LIN {X 0,Y 516.961,Z 452.089,A -85,B 0,C 180,E1 -4941.399,E2 -4941.399} C_VEL
LIN {X 0,Y 517.016,Z 452.086,A -85,B 0,C 180,E1 -4943.757,E2 -4943.757} C_VEL
LIN {X 0,Y 517.09,Z 452.073,A -85,B 0,C 180,E1 -4947.663,E2 -4947.663} C_VEL
LIN {X 0,Y 517.099,Z 452.072,A -85,B 0,C 180,E1 -4950.779,E2 -4950.779} C_VEL
LIN {X 0,Y 517.016,Z 452.086,A -85,B 0,C 180,E1 -4953.117,E2 -4953.117} C_VEL
LIN {X 0,Y 516.993,Z 452.088,A -85,B 0,C 180,E1 -4956.243,E2 -4956.243} C_VEL
LIN {X 0,Y 516.975,Z 452.088,A -85,B 0,C 180,E1 -4958.6,E2 -4958.6} C_VEL
LIN {X 0,Y 516.958,Z 452.09,A -85,B 0,C 180,E1 -4961.807,E2 -4961.807} C_VEL
LIN {X 0,Y 516.951,Z 452.092,A -85,B 0,C 180,E1 -4965.146,E2 -4965.146} C_VEL
LIN {X 0,Y 516.93,Z 452.096,A -85,B 0,C 180,E1 -4968.222,E2 -4968.222} C_VEL
LIN {X 0,Y 516.917,Z 452.093,A -85,B 0,C 180,E1 -4970.701,E2 -4970.701} C_VEL
LIN {X 0,Y 516.909,Z 452.096,A -85,B 0,C 180,E1 -4974.072,E2 -4974.072} C_VEL
LIN {X 0,Y 516.927,Z 452.095,A -85,B 0,C 180,E1 -4976.658,E2 -4976.658} C_VEL
LIN {X 0,Y 516.916,Z 452.1,A -85,B 0,C 180,E1 -4979.523,E2 -4979.523} C_VEL
LIN {X 0,Y 516.9,Z 452.1,A -85,B 0,C 180,E1 -4982.543,E2 -4982.543} C_VEL
LIN {X 0,Y 516.883,Z 452.099,A -85,B 0,C 180,E1 -4985.331,E2 -4985.331} C_VEL
LIN {X 0,Y 516.884,Z 452.099,A -85,B 0,C 180,E1 -4987.943,E2 -4987.943} C_VEL
LIN {X 0,Y 516.886,Z 452.1,A -85,B 0,C 180,E1 -4990.741,E2 -4990.741} C_VEL
LIN {X 0,Y 516.887,Z 452.097,A -85,B 0,C 180,E1 -4992.831,E2 -4992.831} C_VEL
LIN {X 0,Y 516.926,Z 452.097,A -85,B 0,C 180,E1 -4995.01,E2 -4995.01} C_VEL
LIN {X 0,Y 516.919,Z 452.096,A -85,B 0,C 180,E1 -4998.398,E2 -4998.398} C_VEL
LIN {X 0,Y 516.883,Z 452.103,A -85,B 0,C 180,E1 -5001.284,E2 -5001.284} C_VEL
LIN {X 0,Y 516.892,Z 452.102,A -85,B 0,C 180,E1 -5004.221,E2 -5004.221} C_VEL
LIN {X 0,Y 516.899,Z 452.097,A -85,B 0,C 180,E1 -5007.053,E2 -5007.053} C_VEL
LIN {X 0,Y 516.895,Z 452.098,A -85,B 0,C 180,E1 -5009.796,E2 -5009.796} C_VEL
LIN {X 0,Y 516.931,Z 452.095,A -85,B 0,C 180,E1 -5012.467,E2 -5012.467} C_VEL
LIN {X 0,Y 516.911,Z 452.097,A -85,B 0,C 180,E1 -5015.072,E2 -5015.072} C_VEL
LIN {X 0,Y 516.888,Z 452.101,A -85,B 0,C 180,E1 -5018.462,E2 -5018.462} C_VEL
LIN {X 0,Y 516.904,Z 452.096,A -85,B 0,C 180,E1 -5020.955,E2 -5020.955} C_VEL
LIN {X 0,Y 516.916,Z 452.097,A -85,B 0,C 180,E1 -5023.41,E2 -5023.41} C_VEL
LIN {X 0,Y 516.898,Z 452.099,A -85,B 0,C 180,E1 -5025.833,E2 -5025.833} C_VEL
LIN {X 0,Y 516.967,Z 452.088,A -85,B 0,C 180,E1 -5028.233,E2 -5028.233} C_VEL
LIN {X 0,Y 516.971,Z 452.089,A -85,B 0,C 180,E1 -5031.399,E2 -5031.399} C_VEL
LIN {X 0,Y 517.012,Z 452.086,A -85,B 0,C 180,E1 -5033.757,E2 -5033.757} C_VEL
LIN {X 0,Y 517.084,Z 452.075,A -85,B 0,C 180,E1 -5037.663,E2 -5037.663} C_VEL
LIN {X 0,Y 517.095,Z 452.073,A -85,B 0,C 180,E1 -5040.779,E2 -5040.779} C_VEL
LIN {X 0,Y 517.014,Z 452.084,A -85,B 0,C 180,E1 -5043.117,E2 -5043.117} C_VEL
LIN {X 0,Y 517.011,Z 452.086,A -85,B 0,C 180,E1 -5046.243,E2 -5046.243} C_VEL
LIN {X 0,Y 516.952,Z 452.093,A -85,B 0,C 180,E1 -5049.389,E2 -5049.389} C_VEL
LIN {X 0,Y 516.953,Z 452.09,A -85,B 0,C 180,E1 -5051.807,E2 -5051.807} C_VEL
LIN {X 0,Y 516.946,Z 452.091,A -85,B 0,C 180,E1 -5055.146,E2 -5055.146} C_VEL
LIN {X 0,Y 516.926,Z 452.093,A -85,B 0,C 180,E1 -5058.222,E2 -5058.222} C_VEL
LIN {X 0,Y 516.914,Z 452.099,A -85,B 0,C 180,E1 -5060.701,E2 -5060.701} C_VEL
LIN {X 0,Y 516.912,Z 452.095,A -85,B 0,C 180,E1 -5064.072,E2 -5064.072} C_VEL
LIN {X 0,Y 516.927,Z 452.096,A -85,B 0,C 180,E1 -5066.658,E2 -5066.658} C_VEL
LIN {X 0,Y 516.912,Z 452.097,A -85,B 0,C 180,E1 -5069.524,E2 -5069.524} C_VEL
LIN {X 0,Y 516.896,Z 452.097,A -85,B 0,C 180,E1 -5072.543,E2 -5072.543} C_VEL
LIN {X 0,Y 516.882,Z 452.099,A -85,B 0,C 180,E1 -5075.332,E2 -5075.332} C_VEL
LIN {X 0,Y 516.881,Z 452.1,A -85,B 0,C 180,E1 -5077.943,E2 -5077.943} C_VEL
LIN {X 0,Y 516.886,Z 452.102,A -85,B 0,C 180,E1 -5080.742,E2 -5080.742} C_VEL
LIN {X 0,Y 516.906,Z 452.097,A -85,B 0,C 180,E1 -5082.829,E2 -5082.829} C_VEL
LIN {X 0,Y 516.882,Z 452.102,A -85,B 0,C 180,E1 -5086.107,E2 -5086.107} C_VEL
LIN {X 0,Y 516.916,Z 452.1,A -85,B 0,C 180,E1 -5088.399,E2 -5088.399} C_VEL
LIN {X 0,Y 516.905,Z 452.247,A -85,B 0,C 180,E1 -5091.286,E2 -5091.286} C_VEL
LIN {X 0,Y 518.028,Z 458.682,A -85,B 0,C 180,E1 -5093.832,E2 -5093.832} C_VEL
LIN {X 0,Y 518.109,Z 462.545,A -85,B 0,C 180,E1 -5095.27,E2 -5095.27} C_VEL
LIN {X 0,Y 517.824,Z 470.311,A -85,B 0,C 180,E1 -5098.041,E2 -5098.041} C_VEL
LIN {X 0,Y 517.528,Z 478.131,A -85,B 0,C 180,E1 -5100.733,E2 -5100.733} C_VEL
LIN {X 0,Y 517.309,Z 486.015,A -85,B 0,C 180,E1 -5103.364,E2 -5103.364} C_VEL
LIN {X 0,Y 517.111,Z 493.954,A -85,B 0,C 180,E1 -5105.938,E2 -5105.938} C_VEL
LIN {X 0,Y 516.893,Z 503.251,A -85,B 0,C 180,E1 -5108.881,E2 -5108.881} C_VEL
LIN {X 0,Y 516.737,Z 512.695,A -85,B 0,C 180,E1 -5111.771,E2 -5111.771} C_VEL
LIN {X 0,Y 516.643,Z 522.297,A -85,B 0,C 180,E1 -5114.658,E2 -5114.658} C_VEL
LIN {X 0,Y 516.586,Z 527.093,A -85,B 0,C 180,E1 -5116.101,E2 -5116.101} C_VEL
LIN {X 0,Y 518.446,Z 540.212,A -85,B 0,C 180,E1 -5116.452,E2 -5116.452} C_VEL
LIN {X 0,Y 518.207,Z 553.337,A -85,B 0,C 180,E1 -5116.92,E2 -5116.92} C_VEL
LIN {X 0,Y 517.922,Z 565.66,A -85,B 0,C 180,E1 -5117.527,E2 -5117.527} C_VEL
LIN {X 0,Y 517.632,Z 577.009,A -85,B 0,C 180,E1 -5118.249,E2 -5118.249} C_VEL
LIN {X 0,Y 517.298,Z 588.004,A -85,B 0,C 180,E1 -5119.135,E2 -5119.135} C_VEL
LIN {X 0,Y 517.017,Z 596.964,A -85,B 0,C 180,E1 -5120.02,E2 -5120.02} C_VEL
LIN {X 0,Y 516.772,Z 606.702,A -85,B 0,C 180,E1 -5121.199,E2 -5121.199} C_VEL
LIN {X 0,Y 516.562,Z 614.456,A -85,B 0,C 180,E1 -5122.377,E2 -5122.377} C_VEL
LIN {X 0,Y 516.426,Z 621.601,A -85,B 0,C 180,E1 -5123.75,E2 -5123.75} C_VEL
LIN {X 0,Y 516.314,Z 626.35,A -85,B 0,C 180,E1 -5124.924,E2 -5124.924} C_VEL
LIN {X 0,Y 516.354,Z 629.957,A -85,B 0,C 180,E1 -5126.098,E2 -5126.098} C_VEL
LIN {X 0,Y 516.282,Z 631.807,A -85,B 0,C 180,E1 -5126.879,E2 -5126.879} C_VEL
LIN {X 0,Y 516.26,Z 633.192,A -85,B 0,C 180,E1 -5127.66,E2 -5127.66} C_VEL
LIN {X 0,Y 516.16,Z 634.785,A -85,B 0,C 180,E1 -5129.22,E2 -5129.22} C_VEL
LIN {X 0,Y 516.154,Z 635,A -85,B 0,C 180,E1 -5130,E2 -5130} C_VEL
LIN {X 0,Y 516.192,Z 634.183,A -85,B 0,C 180,E1 -5131.561,E2 -5131.561} C_VEL
LIN {X 0,Y 516.26,Z 633.195,A -85,B 0,C 180,E1 -5132.341,E2 -5132.341} C_VEL
LIN {X 0,Y 516.282,Z 631.81,A -85,B 0,C 180,E1 -5133.122,E2 -5133.122} C_VEL
LIN {X 0,Y 516.344,Z 628.89,A -85,B 0,C 180,E1 -5134.293,E2 -5134.293} C_VEL
LIN {X 0,Y 516.405,Z 624.912,A -85,B 0,C 180,E1 -5135.467,E2 -5135.467} C_VEL
LIN {X 0,Y 516.479,Z 618.961,A -85,B 0,C 180,E1 -5136.798,E2 -5136.798} C_VEL
LIN {X 0,Y 516.641,Z 612.011,A -85,B 0,C 180,E1 -5138.015,E2 -5138.015} C_VEL
LIN {X 0,Y 516.844,Z 603.643,A -85,B 0,C 180,E1 -5139.194,E2 -5139.194} C_VEL
LIN {X 0,Y 517.058,Z 595.052,A -85,B 0,C 180,E1 -5140.178,E2 -5140.178} C_VEL
LIN {X 0,Y 517.417,Z 584.448,A -85,B 0,C 180,E1 -5141.161,E2 -5141.161} C_VEL
LIN {X 0,Y 517.697,Z 572.571,A -85,B 0,C 180,E1 -5142.043,E2 -5142.043} C_VEL
LIN {X 0,Y 518.031,Z 560.478,A -85,B 0,C 180,E1 -5142.736,E2 -5142.736} C_VEL
LIN {X 0,Y 518.274,Z 547.989,A -85,B 0,C 180,E1 -5143.278,E2 -5143.278} C_VEL
LIN {X 0,Y 518.222,Z 537.911,A -85,B 0,C 180,E1 -5143.604,E2 -5143.604} C_VEL
LIN {X 0,Y 516.569,Z 526.747,A -85,B 0,C 180,E1 -5143.899,E2 -5143.899} C_VEL
LIN {X 0,Y 516.624,Z 517.508,A -85,B 0,C 180,E1 -5146.6,E2 -5146.6} C_VEL
LIN {X 0,Y 516.753,Z 507.736,A -85,B 0,C 180,E1 -5149.464,E2 -5149.464} C_VEL
LIN {X 0,Y 516.902,Z 498.047,A -85,B 0,C 180,E1 -5152.398,E2 -5152.398} C_VEL
LIN {X 0,Y 517.068,Z 488.591,A -85,B 0,C 180,E1 -5155.35,E2 -5155.35} C_VEL
LIN {X 0,Y 517.247,Z 480.584,A -85,B 0,C 180,E1 -5157.972,E2 -5157.972} C_VEL
LIN {X 0,Y 517.581,Z 471.425,A -85,B 0,C 180,E1 -5161.191,E2 -5161.191} C_VEL
LIN {X 0,Y 517.951,Z 463.912,A -85,B 0,C 180,E1 -5164.137,E2 -5164.137} C_VEL
LIN {X 0,Y 518.131,Z 460.415,A -85,B 0,C 180,E1 -5165.68,E2 -5165.68} C_VEL
LIN {X 0,Y 517.729,Z 456.632,A -85,B 0,C 180,E1 -5167.652,E2 -5167.652} C_VEL
LIN {X 0,Y 517.139,Z 453.466,A -85,B 0,C 180,E1 -5169.698,E2 -5169.698} C_VEL
LIN {X 0,Y 516.906,Z 452.169,A -85,B 0,C 180,E1 -5170.74,E2 -5170.74} C_VEL
LIN {X 0,Y 516.886,Z 452.103,A -85,B 0,C 180,E1 -5173.903,E2 -5173.903} C_VEL
LIN {X 0,Y 516.886,Z 452.103,A -85,B 0,C 180,E1 -5176.107,E2 -5176.107} C_VEL
LIN {X 0,Y 516.921,Z 452.099,A -85,B 0,C 180,E1 -5178.398,E2 -5178.398} C_VEL
LIN {X 0,Y 516.886,Z 452.103,A -85,B 0,C 180,E1 -5181.284,E2 -5181.284} C_VEL
LIN {X 0,Y 516.85,Z 452.296,A -85,B 0,C 180,E1 -5184.218,E2 -5184.218} C_VEL
LIN {X 0,Y 516.898,Z 453.753,A -85,B 0,C 180,E1 -5186.12,E2 -5186.12} C_VEL
LIN {X 0,Y 516.776,Z 456.139,A -85,B 0,C 180,E1 -5188.958,E2 -5188.958} C_VEL
LIN {X 0,Y 516.644,Z 458.463,A -85,B 0,C 180,E1 -5191.568,E2 -5191.568} C_VEL
LIN {X 0,Y 516.58,Z 460.901,A -85,B 0,C 180,E1 -5194.192,E2 -5194.192} C_VEL
LIN {X 0,Y 516.473,Z 463.37,A -85,B 0,C 180,E1 -5196.758,E2 -5196.758} C_VEL
LIN {X 0,Y 516.437,Z 466.473,A -85,B 0,C 180,E1 -5199.884,E2 -5199.884} C_VEL
LIN {X 0,Y 516.371,Z 469.198,A -85,B 0,C 180,E1 -5202.577,E2 -5202.577} C_VEL
LIN {X 0,Y 516.369,Z 471.797,A -85,B 0,C 180,E1 -5205.093,E2 -5205.093} C_VEL
LIN {X 0,Y 516.313,Z 473.008,A -85,B 0,C 180,E1 -5206.219,E2 -5206.219} C_VEL
LIN {X 0,Y 518.436,Z 484.731,A -85,B 0,C 180,E1 -5206.601,E2 -5206.601} C_VEL
LIN {X 0,Y 518.175,Z 497.984,A -85,B 0,C 180,E1 -5207.118,E2 -5207.118} C_VEL
LIN {X 0,Y 517.895,Z 510.399,A -85,B 0,C 180,E1 -5207.785,E2 -5207.785} C_VEL
LIN {X 0,Y 517.609,Z 521.398,A -85,B 0,C 180,E1 -5208.546,E2 -5208.546} C_VEL
LIN {X 0,Y 517.289,Z 531.681,A -85,B 0,C 180,E1 -5209.431,E2 -5209.431} C_VEL
LIN {X 0,Y 517.006,Z 540.914,A -85,B 0,C 180,E1 -5210.414,E2 -5210.414} C_VEL
LIN {X 0,Y 516.778,Z 549.836,A -85,B 0,C 180,E1 -5211.594,E2 -5211.594} C_VEL
LIN {X 0,Y 516.576,Z 557.015,A -85,B 0,C 180,E1 -5212.771,E2 -5212.771} C_VEL
LIN {X 0,Y 516.474,Z 561.855,A -85,B 0,C 180,E1 -5213.75,E2 -5213.75} C_VEL
LIN {X 0,Y 516.314,Z 566.555,A -85,B 0,C 180,E1 -5214.924,E2 -5214.924} C_VEL
LIN {X 0,Y 516.373,Z 570.142,A -85,B 0,C 180,E1 -5216.098,E2 -5216.098} C_VEL
LIN {X 0,Y 516.283,Z 572.001,A -85,B 0,C 180,E1 -5216.879,E2 -5216.879} C_VEL
LIN {X 0,Y 516.261,Z 573.402,A -85,B 0,C 180,E1 -5217.66,E2 -5217.66} C_VEL
LIN {X 0,Y 516.16,Z 575.012,A -85,B 0,C 180,E1 -5219.22,E2 -5219.22} C_VEL
LIN {X 0,Y 516.154,Z 575.245,A -85,B 0,C 180,E1 -5220,E2 -5220} C_VEL
LIN {X 0,Y 516.16,Z 575.06,A -85,B 0,C 180,E1 -5220.78,E2 -5220.78} C_VEL
LIN {X 0,Y 516.261,Z 573.512,A -85,B 0,C 180,E1 -5222.341,E2 -5222.341} C_VEL
LIN {X 0,Y 516.283,Z 572.159,A -85,B 0,C 180,E1 -5223.122,E2 -5223.122} C_VEL
LIN {X 0,Y 516.361,Z 569.301,A -85,B 0,C 180,E1 -5224.293,E2 -5224.293} C_VEL
LIN {X 0,Y 516.4,Z 565.426,A -85,B 0,C 180,E1 -5225.467,E2 -5225.467} C_VEL
LIN {X 0,Y 516.491,Z 559.556,A -85,B 0,C 180,E1 -5226.817,E2 -5226.817} C_VEL
LIN {X 0,Y 516.647,Z 552.886,A -85,B 0,C 180,E1 -5228.015,E2 -5228.015} C_VEL
LIN {X 0,Y 516.846,Z 544.723,A -85,B 0,C 180,E1 -5229.194,E2 -5229.194} C_VEL
LIN {X 0,Y 517.101,Z 536.354,A -85,B 0,C 180,E1 -5230.177,E2 -5230.177} C_VEL
LIN {X 0,Y 517.455,Z 526.003,A -85,B 0,C 180,E1 -5231.16,E2 -5231.16} C_VEL
LIN {X 0,Y 517.737,Z 514.504,A -85,B 0,C 180,E1 -5232.035,E2 -5232.035} C_VEL
LIN {X 0,Y 518.024,Z 502.686,A -85,B 0,C 180,E1 -5232.736,E2 -5232.736} C_VEL
LIN {X 0,Y 518.302,Z 490.589,A -85,B 0,C 180,E1 -5233.278,E2 -5233.278} C_VEL
LIN {X 0,Y 518.282,Z 483.547,A -85,B 0,C 180,E1 -5233.528,E2 -5233.528} C_VEL
LIN {X 0,Y 516.317,Z 472.472,A -85,B 0,C 180,E1 -5233.881,E2 -5233.881} C_VEL
LIN {X 0,Y 516.278,Z 469.363,A -85,B 0,C 180,E1 -5236.611,E2 -5236.611} C_VEL
LIN {X 0,Y 516.319,Z 466.646,A -85,B 0,C 180,E1 -5239.068,E2 -5239.068} C_VEL
LIN {X 0,Y 516.325,Z 463.854,A -85,B 0,C 180,E1 -5241.563,E2 -5241.563} C_VEL
LIN {X 0,Y 516.381,Z 460.895,A -85,B 0,C 180,E1 -5244.233,E2 -5244.233} C_VEL
LIN {X 0,Y 516.432,Z 458.191,A -85,B 0,C 180,E1 -5246.686,E2 -5246.686} C_VEL
LIN {X 0,Y 516.47,Z 455.171,A -85,B 0,C 180,E1 -5249.437,E2 -5249.437} C_VEL
LIN {X 0,Y 516.477,Z 452.324,A -85,B 0,C 180,E1 -5252.053,E2 -5252.053} C_VEL
LIN {X 0,Y 516.805,Z 452.112,A -85,B 0,C 180,E1 -5254.831,E2 -5254.831} C_VEL
LIN {X 0,Y 516.884,Z 452.099,A -85,B 0,C 180,E1 -5257.943,E2 -5257.943} C_VEL
LIN {X 0,Y 516.889,Z 452.098,A -85,B 0,C 180,E1 -5260.742,E2 -5260.742} C_VEL
LIN {X 0,Y 516.884,Z 452.101,A -85,B 0,C 180,E1 -5262.908,E2 -5262.908} C_VEL
LIN {X 0,Y 516.887,Z 452.103,A -85,B 0,C 180,E1 -5266.107,E2 -5266.107} C_VEL
LIN {X 0,Y 516.873,Z 452.102,A -85,B 0,C 180,E1 -5266.304,E2 -5266.304} C_VEL
LIN {X 0,Y 516.197,Z 452.184,A -85,B 0,C 180,E1 -5266.955,E2 -5266.955} C_VEL
LIN {X 0,Y 513.362,Z 452.54,A -85,B 0,C 180,E1 -5268.012,E2 -5268.012} C_VEL
LIN {X 0,Y 510.966,Z 452.84,A -85,B 0,C 180,E1 -5268.864,E2 -5268.864} C_VEL
LIN {X 0,Y 509.926,Z 452.969,A -85,B 0,C 180,E1 -5269.521,E2 -5269.521} C_VEL
LIN {X 0,Y 509.835,Z 452.978,A -85,B 0,C 180,E1 -5269.744,E2 -5269.744} C_VEL
LIN {X 0,Y 509.822,Z 452.98,A -85,B 0,C 180,E1 -5272.659,E2 -5272.659} C_VEL
LIN {X 0,Y 509.862,Z 452.976,A -85,B 0,C 180,E1 -5275.797,E2 -5275.797} C_VEL
LIN {X 0,Y 509.85,Z 452.978,A -85,B 0,C 180,E1 -5278.72,E2 -5278.72} C_VEL
LIN {X 0,Y 509.895,Z 452.974,A -85,B 0,C 180,E1 -5281.901,E2 -5281.901} C_VEL
LIN {X 0,Y 509.882,Z 452.975,A -85,B 0,C 180,E1 -5284.704,E2 -5284.704} C_VEL
LIN {X 0,Y 509.833,Z 452.976,A -85,B 0,C 180,E1 -5287.458,E2 -5287.458} C_VEL
LIN {X 0,Y 509.923,Z 452.969,A -85,B 0,C 180,E1 -5289.845,E2 -5289.845} C_VEL
LIN {X 0,Y 509.885,Z 452.971,A -85,B 0,C 180,E1 -5293.175,E2 -5293.175} C_VEL
LIN {X 0,Y 509.871,Z 452.975,A -85,B 0,C 180,E1 -5295.634,E2 -5295.634} C_VEL
LIN {X 0,Y 509.92,Z 452.969,A -85,B 0,C 180,E1 -5298.874,E2 -5298.874} C_VEL
LIN {X 0,Y 509.927,Z 452.97,A -85,B 0,C 180,E1 -5302.078,E2 -5302.078} C_VEL
LIN {X 0,Y 509.986,Z 452.958,A -85,B 0,C 180,E1 -5304.464,E2 -5304.464} C_VEL
LIN {X 0,Y 510.06,Z 452.949,A -85,B 0,C 180,E1 -5307.631,E2 -5307.631} C_VEL
LIN {X 0,Y 510.07,Z 452.948,A -85,B 0,C 180,E1 -5310.789,E2 -5310.789} C_VEL
LIN {X 0,Y 509.958,Z 452.965,A -85,B 0,C 180,E1 -5313.16,E2 -5313.16} C_VEL
LIN {X 0,Y 509.941,Z 452.965,A -85,B 0,C 180,E1 -5316.33,E2 -5316.33} C_VEL
LIN {X 0,Y 509.921,Z 452.967,A -85,B 0,C 180,E1 -5318.72,E2 -5318.72} C_VEL
LIN {X 0,Y 509.91,Z 452.969,A -85,B 0,C 180,E1 -5321.931,E2 -5321.931} C_VEL
LIN {X 0,Y 509.9,Z 452.971,A -85,B 0,C 180,E1 -5325.241,E2 -5325.241} C_VEL
LIN {X 0,Y 509.887,Z 452.971,A -85,B 0,C 180,E1 -5327.998,E2 -5327.998} C_VEL
LIN {X 0,Y 509.855,Z 452.973,A -85,B 0,C 180,E1 -5331.001,E2 -5331.001} C_VEL
LIN {X 0,Y 509.87,Z 452.975,A -85,B 0,C 180,E1 -5334.426,E2 -5334.426} C_VEL
LIN {X 0,Y 509.887,Z 452.97,A -85,B 0,C 180,E1 -5337.055,E2 -5337.055} C_VEL
LIN {X 0,Y 509.862,Z 452.976,A -85,B 0,C 180,E1 -5339.751,E2 -5339.751} C_VEL
LIN {X 0,Y 509.877,Z 452.974,A -85,B 0,C 180,E1 -5342.774,E2 -5342.774} C_VEL
LIN {X 0,Y 509.843,Z 452.979,A -85,B 0,C 180,E1 -5345.58,E2 -5345.58} C_VEL
LIN {X 0,Y 509.853,Z 452.976,A -85,B 0,C 180,E1 -5348.338,E2 -5348.338} C_VEL
LIN {X 0,Y 509.858,Z 452.974,A -85,B 0,C 180,E1 -5351.425,E2 -5351.425} C_VEL
LIN {X 0,Y 509.86,Z 452.975,A -85,B 0,C 180,E1 -5354.667,E2 -5354.667} C_VEL
LIN {X 0,Y 509.863,Z 452.978,A -85,B 0,C 180,E1 -5358.102,E2 -5358.102} C_VEL
LIN {X 0,Y 509.848,Z 452.975,A -85,B 0,C 180,E1 -5360.647,E2 -5360.647} C_VEL
LIN {X 0,Y 509.838,Z 452.977,A -85,B 0,C 180,E1 -5363.647,E2 -5363.647} C_VEL
LIN {X 0,Y 509.864,Z 452.972,A -85,B 0,C 180,E1 -5366.539,E2 -5366.539} C_VEL
LIN {X 0,Y 509.848,Z 452.978,A -85,B 0,C 180,E1 -5369.334,E2 -5369.334} C_VEL
LIN {X 0,Y 509.897,Z 452.974,A -85,B 0,C 180,E1 -5372.054,E2 -5372.054} C_VEL
LIN {X 0,Y 509.878,Z 452.971,A -85,B 0,C 180,E1 -5374.704,E2 -5374.704} C_VEL
LIN {X 0,Y 509.829,Z 452.979,A -85,B 0,C 180,E1 -5377.458,E2 -5377.458} C_VEL
LIN {X 0,Y 509.919,Z 452.971,A -85,B 0,C 180,E1 -5379.844,E2 -5379.844} C_VEL
LIN {X 0,Y 509.887,Z 452.975,A -85,B 0,C 180,E1 -5383.175,E2 -5383.175} C_VEL
LIN {X 0,Y 509.866,Z 452.974,A -85,B 0,C 180,E1 -5385.634,E2 -5385.634} C_VEL
LIN {X 0,Y 509.915,Z 452.966,A -85,B 0,C 180,E1 -5388.874,E2 -5388.874} C_VEL
LIN {X 0,Y 509.953,Z 452.964,A -85,B 0,C 180,E1 -5392.078,E2 -5392.078} C_VEL
LIN {X 0,Y 509.983,Z 452.959,A -85,B 0,C 180,E1 -5394.464,E2 -5394.464} C_VEL
LIN {X 0,Y 510.055,Z 452.95,A -85,B 0,C 180,E1 -5397.631,E2 -5397.631} C_VEL
LIN {X 0,Y 510.066,Z 452.949,A -85,B 0,C 180,E1 -5400.789,E2 -5400.789} C_VEL
LIN {X 0,Y 509.956,Z 452.964,A -85,B 0,C 180,E1 -5403.16,E2 -5403.16} C_VEL
LIN {X 0,Y 509.98,Z 452.962,A -85,B 0,C 180,E1 -5406.329,E2 -5406.329} C_VEL
LIN {X 0,Y 509.915,Z 452.967,A -85,B 0,C 180,E1 -5408.72,E2 -5408.72} C_VEL
LIN {X 0,Y 509.905,Z 452.968,A -85,B 0,C 180,E1 -5411.932,E2 -5411.932} C_VEL
LIN {X 0,Y 509.895,Z 452.97,A -85,B 0,C 180,E1 -5415.242,E2 -5415.242} C_VEL
LIN {X 0,Y 509.89,Z 452.97,A -85,B 0,C 180,E1 -5418.001,E2 -5418.001} C_VEL
LIN {X 0,Y 509.851,Z 452.976,A -85,B 0,C 180,E1 -5421.002,E2 -5421.002} C_VEL
LIN {X 0,Y 509.871,Z 452.971,A -85,B 0,C 180,E1 -5424.426,E2 -5424.426} C_VEL
LIN {X 0,Y 509.886,Z 452.973,A -85,B 0,C 180,E1 -5427.056,E2 -5427.056} C_VEL
LIN {X 0,Y 509.858,Z 452.979,A -85,B 0,C 180,E1 -5429.751,E2 -5429.751} C_VEL
LIN {X 0,Y 509.874,Z 452.974,A -85,B 0,C 180,E1 -5432.774,E2 -5432.774} C_VEL
LIN {X 0,Y 509.842,Z 452.977,A -85,B 0,C 180,E1 -5435.581,E2 -5435.581} C_VEL
LIN {X 0,Y 509.85,Z 452.974,A -85,B 0,C 180,E1 -5438.338,E2 -5438.338} C_VEL
LIN {X 0,Y 509.859,Z 452.974,A -85,B 0,C 180,E1 -5441.425,E2 -5441.425} C_VEL
LIN {X 0,Y 509.839,Z 452.978,A -85,B 0,C 180,E1 -5444.67,E2 -5444.67} C_VEL
LIN {X 0,Y 509.858,Z 452.977,A -85,B 0,C 180,E1 -5448.103,E2 -5448.103} C_VEL
LIN {X 0,Y 509.885,Z 453.124,A -85,B 0,C 180,E1 -5451.033,E2 -5451.033} C_VEL
LIN {X 0,Y 511.05,Z 459.89,A -85,B 0,C 180,E1 -5453.748,E2 -5453.748} C_VEL
LIN {X 0,Y 511.109,Z 464.798,A -85,B 0,C 180,E1 -5455.592,E2 -5455.592} C_VEL
LIN {X 0,Y 510.796,Z 472.997,A -85,B 0,C 180,E1 -5458.545,E2 -5458.545} C_VEL
LIN {X 0,Y 510.47,Z 480.632,A -85,B 0,C 180,E1 -5461.193,E2 -5461.193} C_VEL
LIN {X 0,Y 510.256,Z 488.504,A -85,B 0,C 180,E1 -5463.848,E2 -5463.848} C_VEL
LIN {X 0,Y 510.009,Z 496.407,A -85,B 0,C 180,E1 -5466.445,E2 -5466.445} C_VEL
LIN {X 0,Y 509.807,Z 506.359,A -85,B 0,C 180,E1 -5469.623,E2 -5469.623} C_VEL
LIN {X 0,Y 509.629,Z 516.437,A -85,B 0,C 180,E1 -5472.753,E2 -5472.753} C_VEL
LIN {X 0,Y 509.494,Z 526.489,A -85,B 0,C 180,E1 -5475.827,E2 -5475.827} C_VEL
LIN {X 0,Y 509.481,Z 526.739,A -85,B 0,C 180,E1 -5475.904,E2 -5475.904} C_VEL
LIN {X 0,Y 511.515,Z 540.496,A -85,B 0,C 180,E1 -5476.29,E2 -5476.29} C_VEL
LIN {X 0,Y 511.273,Z 552.798,A -85,B 0,C 180,E1 -5476.739,E2 -5476.739} C_VEL
LIN {X 0,Y 510.959,Z 565.31,A -85,B 0,C 180,E1 -5477.364,E2 -5477.364} C_VEL
LIN {X 0,Y 510.633,Z 576.491,A -85,B 0,C 180,E1 -5478.086,E2 -5478.086} C_VEL
LIN {X 0,Y 510.29,Z 587.515,A -85,B 0,C 180,E1 -5478.984,E2 -5478.984} C_VEL
LIN {X 0,Y 509.979,Z 596.49,A -85,B 0,C 180,E1 -5479.88,E2 -5479.88} C_VEL
LIN {X 0,Y 509.711,Z 606.242,A -85,B 0,C 180,E1 -5481.077,E2 -5481.077} C_VEL
LIN {X 0,Y 509.494,Z 614.016,A -85,B 0,C 180,E1 -5482.271,E2 -5482.271} C_VEL
LIN {X 0,Y 509.326,Z 621.172,A -85,B 0,C 180,E1 -5483.662,E2 -5483.662} C_VEL
LIN {X 0,Y 509.248,Z 625.934,A -85,B 0,C 180,E1 -5484.854,E2 -5484.854} C_VEL
LIN {X 0,Y 509.268,Z 629.577,A -85,B 0,C 180,E1 -5486.044,E2 -5486.044} C_VEL
LIN {X 0,Y 509.2,Z 631.45,A -85,B 0,C 180,E1 -5486.835,E2 -5486.835} C_VEL
LIN {X 0,Y 509.189,Z 632.857,A -85,B 0,C 180,E1 -5487.627,E2 -5487.627} C_VEL
LIN {X 0,Y 509.073,Z 634.465,A -85,B 0,C 180,E1 -5489.209,E2 -5489.209} C_VEL
LIN {X 0,Y 509.065,Z 634.679,A -85,B 0,C 180,E1 -5490,E2 -5490} C_VEL
LIN {X 0,Y 509.112,Z 633.847,A -85,B 0,C 180,E1 -5491.582,E2 -5491.582} C_VEL
LIN {X 0,Y 509.189,Z 632.846,A -85,B 0,C 180,E1 -5492.373,E2 -5492.373} C_VEL
LIN {X 0,Y 509.2,Z 631.43,A -85,B 0,C 180,E1 -5493.165,E2 -5493.165} C_VEL
LIN {X 0,Y 509.232,Z 628.46,A -85,B 0,C 180,E1 -5494.353,E2 -5494.353} C_VEL
LIN {X 0,Y 509.322,Z 624.44,A -85,B 0,C 180,E1 -5495.543,E2 -5495.543} C_VEL
LIN {X 0,Y 509.402,Z 618.704,A -85,B 0,C 180,E1 -5496.845,E2 -5496.845} C_VEL
LIN {X 0,Y 509.573,Z 611.479,A -85,B 0,C 180,E1 -5498.127,E2 -5498.127} C_VEL
LIN {X 0,Y 509.782,Z 603.072,A -85,B 0,C 180,E1 -5499.323,E2 -5499.323} C_VEL
LIN {X 0,Y 510.031,Z 594.441,A -85,B 0,C 180,E1 -5500.32,E2 -5500.32} C_VEL
LIN {X 0,Y 510.388,Z 583.795,A -85,B 0,C 180,E1 -5501.316,E2 -5501.316} C_VEL
LIN {X 0,Y 510.694,Z 571.873,A -85,B 0,C 180,E1 -5502.211,E2 -5502.211} C_VEL
LIN {X 0,Y 511.046,Z 559.723,A -85,B 0,C 180,E1 -5502.913,E2 -5502.913} C_VEL
LIN {X 0,Y 511.301,Z 547.221,A -85,B 0,C 180,E1 -5503.463,E2 -5503.463} C_VEL
LIN {X 0,Y 511.368,Z 539.322,A -85,B 0,C 180,E1 -5503.728,E2 -5503.728} C_VEL
LIN {X 0,Y 509.474,Z 526.221,A -85,B 0,C 180,E1 -5504.097,E2 -5504.097} C_VEL
LIN {X 0,Y 509.554,Z 517.028,A -85,B 0,C 180,E1 -5506.837,E2 -5506.837} C_VEL
LIN {X 0,Y 509.684,Z 507.317,A -85,B 0,C 180,E1 -5509.745,E2 -5509.745} C_VEL
LIN {X 0,Y 509.858,Z 497.712,A -85,B 0,C 180,E1 -5512.703,E2 -5512.703} C_VEL
LIN {X 0,Y 510.075,Z 488.276,A -85,B 0,C 180,E1 -5515.723,E2 -5515.723} C_VEL
LIN {X 0,Y 510.224,Z 481,A -85,B 0,C 180,E1 -5518.169,E2 -5518.169} C_VEL
LIN {X 0,Y 510.563,Z 473.08,A -85,B 0,C 180,E1 -5521.018,E2 -5521.018} C_VEL
LIN {X 0,Y 510.964,Z 465.954,A -85,B 0,C 180,E1 -5523.853,E2 -5523.853} C_VEL
LIN {X 0,Y 511.166,Z 461.648,A -85,B 0,C 180,E1 -5525.788,E2 -5525.788} C_VEL
LIN {X 0,Y 510.906,Z 458.858,A -85,B 0,C 180,E1 -5527.248,E2 -5527.248} C_VEL
LIN {X 0,Y 510.271,Z 455.297,A -85,B 0,C 180,E1 -5529.53,E2 -5529.53} C_VEL
LIN {X 0,Y 509.87,Z 453.055,A -85,B 0,C 180,E1 -5531.424,E2 -5531.424} C_VEL
LIN {X 0,Y 509.86,Z 452.978,A -85,B 0,C 180,E1 -5534.668,E2 -5534.668} C_VEL
LIN {X 0,Y 509.864,Z 452.977,A -85,B 0,C 180,E1 -5538.103,E2 -5538.103} C_VEL
LIN {X 0,Y 509.851,Z 452.979,A -85,B 0,C 180,E1 -5540.648,E2 -5540.648} C_VEL
LIN {X 0,Y 509.802,Z 453.046,A -85,B 0,C 180,E1 -5543.645,E2 -5543.645} C_VEL
LIN {X 0,Y 509.83,Z 455.143,A -85,B 0,C 180,E1 -5546.537,E2 -5546.537} C_VEL
LIN {X 0,Y 509.725,Z 457.43,A -85,B 0,C 180,E1 -5549.326,E2 -5549.326} C_VEL
LIN {X 0,Y 509.596,Z 459.802,A -85,B 0,C 180,E1 -5552.037,E2 -5552.037} C_VEL
LIN {X 0,Y 509.511,Z 462.229,A -85,B 0,C 180,E1 -5554.685,E2 -5554.685} C_VEL
LIN {X 0,Y 509.409,Z 464.963,A -85,B 0,C 180,E1 -5557.572,E2 -5557.572} C_VEL
LIN {X 0,Y 509.325,Z 468.019,A -85,B 0,C 180,E1 -5560.66,E2 -5560.66} C_VEL
LIN {X 0,Y 509.289,Z 470.549,A -85,B 0,C 180,E1 -5563.155,E2 -5563.155} C_VEL
LIN {X 0,Y 509.295,Z 473.097,A -85,B 0,C 180,E1 -5565.618,E2 -5565.618} C_VEL
LIN {X 0,Y 509.263,Z 473.531,A -85,B 0,C 180,E1 -5566.025,E2 -5566.025} C_VEL
LIN {X 0,Y 511.531,Z 485.645,A -85,B 0,C 180,E1 -5566.442,E2 -5566.442} C_VEL
LIN {X 0,Y 511.275,Z 498.186,A -85,B 0,C 180,E1 -5566.941,E2 -5566.941} C_VEL
LIN {X 0,Y 511.031,Z 509.385,A -85,B 0,C 180,E1 -5567.538,E2 -5567.538} C_VEL
LIN {X 0,Y 510.702,Z 520.401,A -85,B 0,C 180,E1 -5568.289,E2 -5568.289} C_VEL
LIN {X 0,Y 510.326,Z 530.931,A -85,B 0,C 180,E1 -5569.185,E2 -5569.185} C_VEL
LIN {X 0,Y 510.087,Z 539.533,A -85,B 0,C 180,E1 -5570.083,E2 -5570.083} C_VEL
LIN {X 0,Y 509.831,Z 547.446,A -85,B 0,C 180,E1 -5571.079,E2 -5571.079} C_VEL
LIN {X 0,Y 509.579,Z 555.187,A -85,B 0,C 180,E1 -5572.272,E2 -5572.272} C_VEL
LIN {X 0,Y 509.429,Z 562.25,A -85,B 0,C 180,E1 -5573.664,E2 -5573.664} C_VEL
LIN {X 0,Y 509.249,Z 566.961,A -85,B 0,C 180,E1 -5574.854,E2 -5574.854} C_VEL
LIN {X 0,Y 509.303,Z 570.555,A -85,B 0,C 180,E1 -5576.044,E2 -5576.044} C_VEL
LIN {X 0,Y 509.216,Z 572.416,A -85,B 0,C 180,E1 -5576.835,E2 -5576.835} C_VEL
LIN {X 0,Y 509.189,Z 573.819,A -85,B 0,C 180,E1 -5577.627,E2 -5577.627} C_VEL
LIN {X 0,Y 509.074,Z 575.428,A -85,B 0,C 180,E1 -5579.209,E2 -5579.209} C_VEL
LIN {X 0,Y 509.067,Z 575.658,A -85,B 0,C 180,E1 -5580,E2 -5580} C_VEL
LIN {X 0,Y 509.074,Z 575.469,A -85,B 0,C 180,E1 -5580.791,E2 -5580.791} C_VEL
LIN {X 0,Y 509.189,Z 573.909,A -85,B 0,C 180,E1 -5582.373,E2 -5582.373} C_VEL
LIN {X 0,Y 509.202,Z 572.546,A -85,B 0,C 180,E1 -5583.165,E2 -5583.165} C_VEL
LIN {X 0,Y 509.283,Z 569.673,A -85,B 0,C 180,E1 -5584.353,E2 -5584.353} C_VEL
LIN {X 0,Y 509.34,Z 565.78,A -85,B 0,C 180,E1 -5585.543,E2 -5585.543} C_VEL
LIN {X 0,Y 509.455,Z 560.101,A -85,B 0,C 180,E1 -5586.869,E2 -5586.869} C_VEL
LIN {X 0,Y 509.623,Z 553.193,A -85,B 0,C 180,E1 -5588.126,E2 -5588.126} C_VEL
LIN {X 0,Y 509.837,Z 545.001,A -85,B 0,C 180,E1 -5589.322,E2 -5589.322} C_VEL
LIN {X 0,Y 510.108,Z 536.605,A -85,B 0,C 180,E1 -5590.318,E2 -5590.318} C_VEL
LIN {X 0,Y 510.505,Z 526.218,A -85,B 0,C 180,E1 -5591.314,E2 -5591.314} C_VEL
LIN {X 0,Y 510.791,Z 514.695,A -85,B 0,C 180,E1 -5592.201,E2 -5592.201} C_VEL
LIN {X 0,Y 511.093,Z 502.824,A -85,B 0,C 180,E1 -5592.912,E2 -5592.912} C_VEL
LIN {X 0,Y 511.416,Z 489.431,A -85,B 0,C 180,E1 -5593.51,E2 -5593.51} C_VEL
LIN {X 0,Y 511.36,Z 484.397,A -85,B 0,C 180,E1 -5593.689,E2 -5593.689} C_VEL
LIN {X 0,Y 509.236,Z 472.826,A -85,B 0,C 180,E1 -5594.078,E2 -5594.078} C_VEL
LIN {X 0,Y 509.213,Z 469.708,A -85,B 0,C 180,E1 -5596.848,E2 -5596.848} C_VEL
LIN {X 0,Y 509.245,Z 466.92,A -85,B 0,C 180,E1 -5599.343,E2 -5599.343} C_VEL
LIN {X 0,Y 509.29,Z 463.513,A -85,B 0,C 180,E1 -5602.395,E2 -5602.395} C_VEL
LIN {X 0,Y 509.349,Z 460.309,A -85,B 0,C 180,E1 -5605.324,E2 -5605.324} C_VEL
LIN {X 0,Y 509.368,Z 457.36,A -85,B 0,C 180,E1 -5607.988,E2 -5607.988} C_VEL
LIN {X 0,Y 509.397,Z 454.426,A -85,B 0,C 180,E1 -5610.696,E2 -5610.696} C_VEL
LIN {X 0,Y 509.403,Z 453.441,A -85,B 0,C 180,E1 -5611.619,E2 -5611.619} C_VEL
LIN {X 0,Y 509.485,Z 453.025,A -85,B 0,C 180,E1 -5612.706,E2 -5612.706} C_VEL
LIN {X 0,Y 509.775,Z 452.987,A -85,B 0,C 180,E1 -5615.383,E2 -5615.383} C_VEL
LIN {X 0,Y 509.854,Z 452.979,A -85,B 0,C 180,E1 -5618.338,E2 -5618.338} C_VEL
LIN {X 0,Y 509.862,Z 452.976,A -85,B 0,C 180,E1 -5621.425,E2 -5621.425} C_VEL
LIN {X 0,Y 509.844,Z 452.979,A -85,B 0,C 180,E1 -5624.67,E2 -5624.67} C_VEL
LIN {X 0,Y 509.861,Z 452.976,A -85,B 0,C 180,E1 -5628.103,E2 -5628.103} C_VEL
LIN {X 0,Y 509.835,Z 452.978,A -85,B 0,C 180,E1 -5629.744,E2 -5629.744} C_VEL
LIN {X 0,Y 509.153,Z 453.065,A -85,B 0,C 180,E1 -5630.403,E2 -5630.403} C_VEL
LIN {X 0,Y 506.305,Z 453.417,A -85,B 0,C 180,E1 -5631.475,E2 -5631.475} C_VEL
LIN {X 0,Y 503.9,Z 453.721,A -85,B 0,C 180,E1 -5632.338,E2 -5632.338} C_VEL
LIN {X 0,Y 502.858,Z 453.845,A -85,B 0,C 180,E1 -5633.004,E2 -5633.004} C_VEL
LIN {X 0,Y 502.767,Z 453.855,A -85,B 0,C 180,E1 -5633.23,E2 -5633.23} C_VEL
LIN {X 0,Y 502.81,Z 453.853,A -85,B 0,C 180,E1 -5636.006,E2 -5636.006} C_VEL
LIN {X 0,Y 502.8,Z 453.855,A -85,B 0,C 180,E1 -5638.857,E2 -5638.857} C_VEL
LIN {X 0,Y 502.846,Z 453.85,A -85,B 0,C 180,E1 -5641.706,E2 -5641.706} C_VEL
LIN {X 0,Y 502.846,Z 453.849,A -85,B 0,C 180,E1 -5644.324,E2 -5644.324} C_VEL
LIN {X 0,Y 502.81,Z 453.851,A -85,B 0,C 180,E1 -5647.297,E2 -5647.297} C_VEL
LIN {X 0,Y 502.83,Z 453.85,A -85,B 0,C 180,E1 -5650.4,E2 -5650.4} C_VEL
LIN {X 0,Y 502.834,Z 453.851,A -85,B 0,C 180,E1 -5652.931,E2 -5652.931} C_VEL
LIN {X 0,Y 502.852,Z 453.847,A -85,B 0,C 180,E1 -5655.429,E2 -5655.429} C_VEL
LIN {X 0,Y 502.884,Z 453.846,A -85,B 0,C 180,E1 -5658.717,E2 -5658.717} C_VEL
LIN {X 0,Y 502.886,Z 453.847,A -85,B 0,C 180,E1 -5661.966,E2 -5661.966} C_VEL
LIN {X 0,Y 502.942,Z 453.836,A -85,B 0,C 180,E1 -5664.386,E2 -5664.386} C_VEL
LIN {X 0,Y 503.03,Z 453.825,A -85,B 0,C 180,E1 -5667.598,E2 -5667.598} C_VEL
LIN {X 0,Y 503.034,Z 453.827,A -85,B 0,C 180,E1 -5670,E2 -5670} C_VEL
LIN {X 0,Y 503.03,Z 453.826,A -85,B 0,C 180,E1 -5672.402,E2 -5672.402} C_VEL
LIN {X 0,Y 502.932,Z 453.837,A -85,B 0,C 180,E1 -5675.613,E2 -5675.613} C_VEL
LIN {X 0,Y 502.88,Z 453.845,A -85,B 0,C 180,E1 -5678.843,E2 -5678.843} C_VEL
LIN {X 0,Y 502.852,Z 453.85,A -85,B 0,C 180,E1 -5682.101,E2 -5682.101} C_VEL
LIN {X 0,Y 502.854,Z 453.85,A -85,B 0,C 180,E1 -5685.399,E2 -5685.399} C_VEL
LIN {X 0,Y 502.846,Z 453.849,A -85,B 0,C 180,E1 -5688.12,E2 -5688.12} C_VEL
LIN {X 0,Y 502.834,Z 453.848,A -85,B 0,C 180,E1 -5690.536,E2 -5690.536} C_VEL
LIN {X 0,Y 502.796,Z 453.856,A -85,B 0,C 180,E1 -5693.04,E2 -5693.04} C_VEL
LIN {X 0,Y 502.844,Z 453.848,A -85,B 0,C 180,E1 -5695.675,E2 -5695.675} C_VEL
LIN {X 0,Y 502.844,Z 453.848,A -85,B 0,C 180,E1 -5698.372,E2 -5698.372} C_VEL
LIN {X 0,Y 502.797,Z 453.855,A -85,B 0,C 180,E1 -5701.498,E2 -5701.498} C_VEL
LIN {X 0,Y 502.809,Z 453.853,A -85,B 0,C 180,E1 -5704.444,E2 -5704.444} C_VEL
LIN {X 0,Y 502.784,Z 453.858,A -85,B 0,C 180,E1 -5707.178,E2 -5707.178} C_VEL
LIN {X 0,Y 502.791,Z 453.857,A -85,B 0,C 180,E1 -5710.015,E2 -5710.015} C_VEL
LIN {X 0,Y 502.806,Z 453.853,A -85,B 0,C 180,E1 -5712.199,E2 -5712.199} C_VEL
LIN {X 0,Y 502.804,Z 453.854,A -85,B 0,C 180,E1 -5715.468,E2 -5715.468} C_VEL
LIN {X 0,Y 502.833,Z 453.852,A -85,B 0,C 180,E1 -5717.864,E2 -5717.864} C_VEL
LIN {X 0,Y 502.804,Z 453.854,A -85,B 0,C 180,E1 -5721.024,E2 -5721.024} C_VEL
LIN {X 0,Y 502.787,Z 453.858,A -85,B 0,C 180,E1 -5724.167,E2 -5724.167} C_VEL
LIN {X 0,Y 502.835,Z 453.848,A -85,B 0,C 180,E1 -5726.993,E2 -5726.993} C_VEL
LIN {X 0,Y 502.817,Z 453.852,A -85,B 0,C 180,E1 -5730.065,E2 -5730.065} C_VEL
LIN {X 0,Y 502.836,Z 453.85,A -85,B 0,C 180,E1 -5732.533,E2 -5732.533} C_VEL
LIN {X 0,Y 502.829,Z 453.853,A -85,B 0,C 180,E1 -5735.299,E2 -5735.299} C_VEL
LIN {X 0,Y 502.782,Z 453.856,A -85,B 0,C 180,E1 -5737.826,E2 -5737.826} C_VEL
LIN {X 0,Y 502.827,Z 453.85,A -85,B 0,C 180,E1 -5740.4,E2 -5740.4} C_VEL
LIN {X 0,Y 502.836,Z 453.851,A -85,B 0,C 180,E1 -5742.931,E2 -5742.931} C_VEL
LIN {X 0,Y 502.847,Z 453.848,A -85,B 0,C 180,E1 -5745.429,E2 -5745.429} C_VEL
LIN {X 0,Y 502.879,Z 453.842,A -85,B 0,C 180,E1 -5748.717,E2 -5748.717} C_VEL
LIN {X 0,Y 502.904,Z 453.842,A -85,B 0,C 180,E1 -5751.966,E2 -5751.966} C_VEL
LIN {X 0,Y 502.939,Z 453.837,A -85,B 0,C 180,E1 -5754.386,E2 -5754.386} C_VEL
LIN {X 0,Y 503.025,Z 453.826,A -85,B 0,C 180,E1 -5757.598,E2 -5757.598} C_VEL
LIN {X 0,Y 503.029,Z 453.828,A -85,B 0,C 180,E1 -5760,E2 -5760} C_VEL
LIN {X 0,Y 503.025,Z 453.824,A -85,B 0,C 180,E1 -5762.402,E2 -5762.402} C_VEL
LIN {X 0,Y 502.939,Z 453.836,A -85,B 0,C 180,E1 -5765.613,E2 -5765.613} C_VEL
LIN {X 0,Y 502.903,Z 453.844,A -85,B 0,C 180,E1 -5768.033,E2 -5768.033} C_VEL
LIN {X 0,Y 502.878,Z 453.848,A -85,B 0,C 180,E1 -5771.283,E2 -5771.283} C_VEL
LIN {X 0,Y 502.846,Z 453.85,A -85,B 0,C 180,E1 -5774.571,E2 -5774.571} C_VEL
LIN {X 0,Y 502.863,Z 453.845,A -85,B 0,C 180,E1 -5777.907,E2 -5777.907} C_VEL
LIN {X 0,Y 502.83,Z 453.852,A -85,B 0,C 180,E1 -5780.536,E2 -5780.536} C_VEL
LIN {X 0,Y 502.795,Z 453.854,A -85,B 0,C 180,E1 -5783.04,E2 -5783.04} C_VEL
LIN {X 0,Y 502.841,Z 453.849,A -85,B 0,C 180,E1 -5785.675,E2 -5785.675} C_VEL
LIN {X 0,Y 502.841,Z 453.851,A -85,B 0,C 180,E1 -5788.373,E2 -5788.373} C_VEL
LIN {X 0,Y 502.793,Z 453.858,A -85,B 0,C 180,E1 -5791.499,E2 -5791.499} C_VEL
LIN {X 0,Y 502.806,Z 453.855,A -85,B 0,C 180,E1 -5794.444,E2 -5794.444} C_VEL
LIN {X 0,Y 502.782,Z 453.857,A -85,B 0,C 180,E1 -5797.178,E2 -5797.178} C_VEL
LIN {X 0,Y 502.789,Z 453.854,A -85,B 0,C 180,E1 -5800.015,E2 -5800.015} C_VEL
LIN {X 0,Y 502.831,Z 453.852,A -85,B 0,C 180,E1 -5802.203,E2 -5802.203} C_VEL
LIN {X 0,Y 502.78,Z 453.862,A -85,B 0,C 180,E1 -5805.66,E2 -5805.66} C_VEL
LIN {X 0,Y 502.82,Z 453.854,A -85,B 0,C 180,E1 -5809.005,E2 -5809.005} C_VEL
LIN {X 0,Y 502.835,Z 453.988,A -85,B 0,C 180,E1 -5810.769,E2 -5810.769} C_VEL
LIN {X 0,Y 504.032,Z 460.911,A -85,B 0,C 180,E1 -5813.597,E2 -5813.597} C_VEL
LIN {X 0,Y 504.203,Z 464.947,A -85,B 0,C 180,E1 -5815.146,E2 -5815.146} C_VEL
LIN {X 0,Y 503.836,Z 473.571,A -85,B 0,C 180,E1 -5818.309,E2 -5818.309} C_VEL
LIN {X 0,Y 503.455,Z 481.796,A -85,B 0,C 180,E1 -5821.21,E2 -5821.21} C_VEL
LIN {X 0,Y 503.218,Z 489.643,A -85,B 0,C 180,E1 -5823.901,E2 -5823.901} C_VEL
LIN {X 0,Y 502.959,Z 497.549,A -85,B 0,C 180,E1 -5826.532,E2 -5826.532} C_VEL
LIN {X 0,Y 502.755,Z 506.82,A -85,B 0,C 180,E1 -5829.545,E2 -5829.545} C_VEL
LIN {X 0,Y 502.568,Z 516.119,A -85,B 0,C 180,E1 -5832.503,E2 -5832.503} C_VEL
LIN {X 0,Y 502.433,Z 525.469,A -85,B 0,C 180,E1 -5835.417,E2 -5835.417} C_VEL
LIN {X 0,Y 502.403,Z 526.387,A -85,B 0,C 180,E1 -5835.701,E2 -5835.701} C_VEL
LIN {X 0,Y 504.546,Z 540.744,A -85,B 0,C 180,E1 -5836.123,E2 -5836.123} C_VEL
LIN {X 0,Y 504.307,Z 553.392,A -85,B 0,C 180,E1 -5836.604,E2 -5836.604} C_VEL
LIN {X 0,Y 503.969,Z 566.214,A -85,B 0,C 180,E1 -5837.27,E2 -5837.27} C_VEL
LIN {X 0,Y 503.597,Z 577.333,A -85,B 0,C 180,E1 -5838.019,E2 -5838.019} C_VEL
LIN {X 0,Y 503.238,Z 588.104,A -85,B 0,C 180,E1 -5838.929,E2 -5838.929} C_VEL
LIN {X 0,Y 502.887,Z 597.81,A -85,B 0,C 180,E1 -5839.939,E2 -5839.939} C_VEL
LIN {X 0,Y 502.661,Z 605.782,A -85,B 0,C 180,E1 -5840.95,E2 -5840.95} C_VEL
LIN {X 0,Y 502.416,Z 613.576,A -85,B 0,C 180,E1 -5842.161,E2 -5842.161} C_VEL
LIN {X 0,Y 502.228,Z 620.368,A -85,B 0,C 180,E1 -5843.49,E2 -5843.49} C_VEL
LIN {X 0,Y 502.183,Z 625.517,A -85,B 0,C 180,E1 -5844.781,E2 -5844.781} C_VEL
LIN {X 0,Y 502.165,Z 629.165,A -85,B 0,C 180,E1 -5845.988,E2 -5845.988} C_VEL
LIN {X 0,Y 502.121,Z 631.043,A -85,B 0,C 180,E1 -5846.791,E2 -5846.791} C_VEL
LIN {X 0,Y 502.12,Z 632.453,A -85,B 0,C 180,E1 -5847.594,E2 -5847.594} C_VEL
LIN {X 0,Y 501.99,Z 634.059,A -85,B 0,C 180,E1 -5849.198,E2 -5849.198} C_VEL
LIN {X 0,Y 501.98,Z 634.27,A -85,B 0,C 180,E1 -5850,E2 -5850} C_VEL
LIN {X 0,Y 502.036,Z 633.431,A -85,B 0,C 180,E1 -5851.605,E2 -5851.605} C_VEL
LIN {X 0,Y 502.12,Z 632.422,A -85,B 0,C 180,E1 -5852.407,E2 -5852.407} C_VEL
LIN {X 0,Y 502.121,Z 630.994,A -85,B 0,C 180,E1 -5853.21,E2 -5853.21} C_VEL
LIN {X 0,Y 502.127,Z 628.005,A -85,B 0,C 180,E1 -5854.415,E2 -5854.415} C_VEL
LIN {X 0,Y 502.238,Z 623.965,A -85,B 0,C 180,E1 -5855.622,E2 -5855.622} C_VEL
LIN {X 0,Y 502.332,Z 617.844,A -85,B 0,C 180,E1 -5857.012,E2 -5857.012} C_VEL
LIN {X 0,Y 502.499,Z 610.946,A -85,B 0,C 180,E1 -5858.242,E2 -5858.242} C_VEL
LIN {X 0,Y 502.728,Z 602.5,A -85,B 0,C 180,E1 -5859.455,E2 -5859.455} C_VEL
LIN {X 0,Y 503.013,Z 593.828,A -85,B 0,C 180,E1 -5860.465,E2 -5860.465} C_VEL
LIN {X 0,Y 503.342,Z 583.14,A -85,B 0,C 180,E1 -5861.477,E2 -5861.477} C_VEL
LIN {X 0,Y 503.672,Z 572.162,A -85,B 0,C 180,E1 -5862.315,E2 -5862.315} C_VEL
LIN {X 0,Y 504.06,Z 559.973,A -85,B 0,C 180,E1 -5863.044,E2 -5863.044} C_VEL
LIN {X 0,Y 504.379,Z 546.459,A -85,B 0,C 180,E1 -5863.651,E2 -5863.651} C_VEL
LIN {X 0,Y 504.379,Z 539.871,A -85,B 0,C 180,E1 -5863.882,E2 -5863.882} C_VEL
LIN {X 0,Y 502.551,Z 527.372,A -85,B 0,C 180,E1 -5864.247,E2 -5864.247} C_VEL
LIN {X 0,Y 502.388,Z 525.696,A -85,B 0,C 180,E1 -5864.3,E2 -5864.3} C_VEL
LIN {X 0,Y 502.476,Z 516.495,A -85,B 0,C 180,E1 -5867.081,E2 -5867.081} C_VEL
LIN {X 0,Y 502.692,Z 505.494,A -85,B 0,C 180,E1 -5870.458,E2 -5870.458} C_VEL
LIN {X 0,Y 502.831,Z 495.97,A -85,B 0,C 180,E1 -5873.475,E2 -5873.475} C_VEL
LIN {X 0,Y 503.053,Z 486.532,A -85,B 0,C 180,E1 -5876.603,E2 -5876.603} C_VEL
LIN {X 0,Y 503.273,Z 478.985,A -85,B 0,C 180,E1 -5879.259,E2 -5879.259} C_VEL
LIN {X 0,Y 503.622,Z 472.644,A -85,B 0,C 180,E1 -5881.652,E2 -5881.652} C_VEL
LIN {X 0,Y 503.988,Z 467.187,A -85,B 0,C 180,E1 -5883.903,E2 -5883.903} C_VEL
LIN {X 0,Y 504.199,Z 462.566,A -85,B 0,C 180,E1 -5886.054,E2 -5886.054} C_VEL
LIN {X 0,Y 503.793,Z 459.338,A -85,B 0,C 180,E1 -5887.866,E2 -5887.866} C_VEL
LIN {X 0,Y 503.238,Z 456.302,A -85,B 0,C 180,E1 -5889.972,E2 -5889.972} C_VEL
LIN {X 0,Y 502.833,Z 453.952,A -85,B 0,C 180,E1 -5892.203,E2 -5892.203} C_VEL
LIN {X 0,Y 502.804,Z 453.857,A -85,B 0,C 180,E1 -5895.468,E2 -5895.468} C_VEL
LIN {X 0,Y 502.833,Z 453.853,A -85,B 0,C 180,E1 -5897.864,E2 -5897.864} C_VEL
LIN {X 0,Y 502.806,Z 453.857,A -85,B 0,C 180,E1 -5901.024,E2 -5901.024} C_VEL
LIN {X 0,Y 502.755,Z 453.877,A -85,B 0,C 180,E1 -5903.052,E2 -5903.052} C_VEL
LIN {X 0,Y 502.856,Z 455.487,A -85,B 0,C 180,E1 -5905.548,E2 -5905.548} C_VEL
LIN {X 0,Y 502.729,Z 457.755,A -85,B 0,C 180,E1 -5908.514,E2 -5908.514} C_VEL
LIN {X 0,Y 502.589,Z 460.472,A -85,B 0,C 180,E1 -5911.76,E2 -5911.76} C_VEL
LIN {X 0,Y 502.482,Z 462.752,A -85,B 0,C 180,E1 -5914.305,E2 -5914.305} C_VEL
LIN {X 0,Y 502.371,Z 465.645,A -85,B 0,C 180,E1 -5917.417,E2 -5917.417} C_VEL
LIN {X 0,Y 502.274,Z 468.517,A -85,B 0,C 180,E1 -5920.378,E2 -5920.378} C_VEL
LIN {X 0,Y 502.241,Z 471.053,A -85,B 0,C 180,E1 -5922.911,E2 -5922.911} C_VEL
LIN {X 0,Y 502.223,Z 474.102,A -85,B 0,C 180,E1 -5925.851,E2 -5925.851} C_VEL
LIN {X 0,Y 504.358,Z 484.724,A -85,B 0,C 180,E1 -5926.207,E2 -5926.207} C_VEL
LIN {X 0,Y 504.579,Z 488.757,A -85,B 0,C 180,E1 -5926.355,E2 -5926.355} C_VEL
LIN {X 0,Y 504.297,Z 501.481,A -85,B 0,C 180,E1 -5926.911,E2 -5926.911} C_VEL
LIN {X 0,Y 503.981,Z 513.51,A -85,B 0,C 180,E1 -5927.612,E2 -5927.612} C_VEL
LIN {X 0,Y 503.634,Z 524.495,A -85,B 0,C 180,E1 -5928.428,E2 -5928.428} C_VEL
LIN {X 0,Y 503.291,Z 534.306,A -85,B 0,C 180,E1 -5929.338,E2 -5929.338} C_VEL
LIN {X 0,Y 502.99,Z 543.217,A -85,B 0,C 180,E1 -5930.348,E2 -5930.348} C_VEL
LIN {X 0,Y 502.703,Z 551.907,A -85,B 0,C 180,E1 -5931.559,E2 -5931.559} C_VEL
LIN {X 0,Y 502.468,Z 558.831,A -85,B 0,C 180,E1 -5932.768,E2 -5932.768} C_VEL
LIN {X 0,Y 502.362,Z 564.351,A -85,B 0,C 180,E1 -5933.977,E2 -5933.977} C_VEL
LIN {X 0,Y 502.138,Z 568.69,A -85,B 0,C 180,E1 -5935.183,E2 -5935.183} C_VEL
LIN {X 0,Y 502.236,Z 570.967,A -85,B 0,C 180,E1 -5935.988,E2 -5935.988} C_VEL
LIN {X 0,Y 502.137,Z 572.831,A -85,B 0,C 180,E1 -5936.791,E2 -5936.791} C_VEL
LIN {X 0,Y 502.121,Z 574.237,A -85,B 0,C 180,E1 -5937.594,E2 -5937.594} C_VEL
LIN {X 0,Y 501.991,Z 575.843,A -85,B 0,C 180,E1 -5939.198,E2 -5939.198} C_VEL
LIN {X 0,Y 501.982,Z 576.07,A -85,B 0,C 180,E1 -5940,E2 -5940} C_VEL
LIN {X 0,Y 501.991,Z 575.877,A -85,B 0,C 180,E1 -5940.802,E2 -5940.802} C_VEL
LIN {X 0,Y 502.12,Z 574.302,A -85,B 0,C 180,E1 -5942.407,E2 -5942.407} C_VEL
LIN {X 0,Y 502.125,Z 572.933,A -85,B 0,C 180,E1 -5943.21,E2 -5943.21} C_VEL
LIN {X 0,Y 502.209,Z 570.045,A -85,B 0,C 180,E1 -5944.415,E2 -5944.415} C_VEL
LIN {X 0,Y 502.283,Z 566.134,A -85,B 0,C 180,E1 -5945.621,E2 -5945.621} C_VEL
LIN {X 0,Y 502.391,Z 561.088,A -85,B 0,C 180,E1 -5946.829,E2 -5946.829} C_VEL
LIN {X 0,Y 502.554,Z 554.721,A -85,B 0,C 180,E1 -5948.039,E2 -5948.039} C_VEL
LIN {X 0,Y 502.768,Z 546.766,A -85,B 0,C 180,E1 -5949.251,E2 -5949.251} C_VEL
LIN {X 0,Y 503.095,Z 538.642,A -85,B 0,C 180,E1 -5950.26,E2 -5950.26} C_VEL
LIN {X 0,Y 503.451,Z 528.735,A -85,B 0,C 180,E1 -5951.27,E2 -5951.27} C_VEL
LIN {X 0,Y 503.818,Z 517.607,A -85,B 0,C 180,E1 -5952.176,E2 -5952.176} C_VEL
LIN {X 0,Y 504.092,Z 506.616,A -85,B 0,C 180,E1 -5952.89,E2 -5952.89} C_VEL
LIN {X 0,Y 504.425,Z 494.57,A -85,B 0,C 180,E1 -5953.496,E2 -5953.496} C_VEL
LIN {X 0,Y 504.477,Z 485.614,A -85,B 0,C 180,E1 -5953.841,E2 -5953.841} C_VEL
LIN {X 0,Y 502.463,Z 474.698,A -85,B 0,C 180,E1 -5954.213,E2 -5954.213} C_VEL
LIN {X 0,Y 502.173,Z 473.165,A -85,B 0,C 180,E1 -5954.281,E2 -5954.281} C_VEL
LIN {X 0,Y 502.182,Z 469.049,A -85,B 0,C 180,E1 -5957.932,E2 -5957.932} C_VEL
LIN {X 0,Y 502.175,Z 466.214,A -85,B 0,C 180,E1 -5960.48,E2 -5960.48} C_VEL
LIN {X 0,Y 502.194,Z 463.363,A -85,B 0,C 180,E1 -5963.07,E2 -5963.07} C_VEL
LIN {X 0,Y 502.271,Z 460.465,A -85,B 0,C 180,E1 -5965.707,E2 -5965.707} C_VEL
LIN {X 0,Y 502.304,Z 457.531,A -85,B 0,C 180,E1 -5968.406,E2 -5968.406} C_VEL
LIN {X 0,Y 502.332,Z 454.304,A -85,B 0,C 180,E1 -5971.412,E2 -5971.412} C_VEL
LIN {X 0,Y 502.376,Z 453.91,A -85,B 0,C 180,E1 -5972.114,E2 -5972.114} C_VEL
LIN {X 0,Y 502.686,Z 453.871,A -85,B 0,C 180,E1 -5974.975,E2 -5974.975} C_VEL
LIN {X 0,Y 502.795,Z 453.855,A -85,B 0,C 180,E1 -5977.954,E2 -5977.954} C_VEL
LIN {X 0,Y 502.825,Z 453.851,A -85,B 0,C 180,E1 -5981.066,E2 -5981.066} C_VEL
LIN {X 0,Y 502.791,Z 453.859,A -85,B 0,C 180,E1 -5984.53,E2 -5984.53} C_VEL
LIN {X 0,Y 502.8,Z 453.858,A -85,B 0,C 180,E1 -5987.861,E2 -5987.861} C_VEL
LIN {X 0,Y 502.807,Z 453.854,A -85,B 0,C 180,E1 -5991.024,E2 -5991.024} C_VEL
LIN {X 0,Y 502.767,Z 453.855,A -85,B 0,C 180,E1 -5993.23,E2 -5993.23} C_VEL
LIN {X 0,Y 502.102,Z 453.943,A -85,B 0,C 180,E1 -5993.899,E2 -5993.899} C_VEL
LIN {X 0,Y 499.306,Z 454.292,A -85,B 0,C 180,E1 -5994.986,E2 -5994.986} C_VEL
LIN {X 0,Y 496.934,Z 454.589,A -85,B 0,C 180,E1 -5995.862,E2 -5995.862} C_VEL
LIN {X 0,Y 495.894,Z 454.717,A -85,B 0,C 180,E1 -5996.538,E2 -5996.538} C_VEL
LIN {X 0,Y 495.797,Z 454.728,A -85,B 0,C 180,E1 -5996.767,E2 -5996.767} C_VEL
LIN {X 0,Y 495.769,Z 454.73,A -85,B 0,C 180,E1 -5999.853,E2 -5999.853} C_VEL
LIN {X 0,Y 495.818,Z 454.725,A -85,B 0,C 180,E1 -6003.026,E2 -6003.026} C_VEL
LIN {X 0,Y 495.754,Z 454.731,A -85,B 0,C 180,E1 -6005.725,E2 -6005.725} C_VEL
LIN {X 0,Y 495.749,Z 454.733,A -85,B 0,C 180,E1 -6008.371,E2 -6008.371} C_VEL
LIN {X 0,Y 495.79,Z 454.729,A -85,B 0,C 180,E1 -6010.972,E2 -6010.972} C_VEL
LIN {X 0,Y 495.782,Z 454.727,A -85,B 0,C 180,E1 -6013.53,E2 -6013.53} C_VEL
LIN {X 0,Y 495.8,Z 454.728,A -85,B 0,C 180,E1 -6016.056,E2 -6016.056} C_VEL
LIN {X 0,Y 495.858,Z 454.72,A -85,B 0,C 180,E1 -6018.555,E2 -6018.555} C_VEL
LIN {X 0,Y 495.842,Z 454.723,A -85,B 0,C 180,E1 -6021.851,E2 -6021.851} C_VEL
LIN {X 0,Y 495.9,Z 454.713,A -85,B 0,C 180,E1 -6024.306,E2 -6024.306} C_VEL
LIN {X 0,Y 495.999,Z 454.7,A -85,B 0,C 180,E1 -6027.564,E2 -6027.564} C_VEL
LIN {X 0,Y 496.011,Z 454.699,A -85,B 0,C 180,E1 -6030.812,E2 -6030.812} C_VEL
LIN {X 0,Y 495.845,Z 454.722,A -85,B 0,C 180,E1 -6033.25,E2 -6033.25} C_VEL
LIN {X 0,Y 495.843,Z 454.72,A -85,B 0,C 180,E1 -6036.511,E2 -6036.511} C_VEL
LIN {X 0,Y 495.848,Z 454.721,A -85,B 0,C 180,E1 -6038.969,E2 -6038.969} C_VEL
LIN {X 0,Y 495.834,Z 454.724,A -85,B 0,C 180,E1 -6042.035,E2 -6042.035} C_VEL
LIN {X 0,Y 495.829,Z 454.725,A -85,B 0,C 180,E1 -6045.451,E2 -6045.451} C_VEL
LIN {X 0,Y 495.812,Z 454.727,A -85,B 0,C 180,E1 -6048.247,E2 -6048.247} C_VEL
LIN {X 0,Y 495.779,Z 454.726,A -85,B 0,C 180,E1 -6050.756,E2 -6050.756} C_VEL
LIN {X 0,Y 495.753,Z 454.735,A -85,B 0,C 180,E1 -6053.387,E2 -6053.387} C_VEL
LIN {X 0,Y 495.795,Z 454.729,A -85,B 0,C 180,E1 -6056.067,E2 -6056.067} C_VEL
LIN {X 0,Y 495.776,Z 454.727,A -85,B 0,C 180,E1 -6058.814,E2 -6058.814} C_VEL
LIN {X 0,Y 495.759,Z 454.731,A -85,B 0,C 180,E1 -6061.725,E2 -6061.725} C_VEL
LIN {X 0,Y 495.779,Z 454.727,A -85,B 0,C 180,E1 -6064.695,E2 -6064.695} C_VEL
LIN {X 0,Y 495.735,Z 454.736,A -85,B 0,C 180,E1 -6067.561,E2 -6067.561} C_VEL
LIN {X 0,Y 495.769,Z 454.73,A -85,B 0,C 180,E1 -6070.7,E2 -6070.7} C_VEL
LIN {X 0,Y 495.737,Z 454.734,A -85,B 0,C 180,E1 -6074,E2 -6074} C_VEL
LIN {X 0,Y 495.737,Z 454.734,A -85,B 0,C 180,E1 -6077.117,E2 -6077.117} C_VEL
LIN {X 0,Y 495.761,Z 454.732,A -85,B 0,C 180,E1 -6079.953,E2 -6079.953} C_VEL
LIN {X 0,Y 495.733,Z 454.736,A -85,B 0,C 180,E1 -6082.552,E2 -6082.552} C_VEL
LIN {X 0,Y 495.786,Z 454.728,A -85,B 0,C 180,E1 -6085.457,E2 -6085.457} C_VEL
LIN {X 0,Y 495.759,Z 454.73,A -85,B 0,C 180,E1 -6088.364,E2 -6088.364} C_VEL
LIN {X 0,Y 495.79,Z 454.727,A -85,B 0,C 180,E1 -6091.506,E2 -6091.506} C_VEL
LIN {X 0,Y 495.793,Z 454.728,A -85,B 0,C 180,E1 -6093.932,E2 -6093.932} C_VEL
LIN {X 0,Y 495.762,Z 454.733,A -85,B 0,C 180,E1 -6097.139,E2 -6097.139} C_VEL
LIN {X 0,Y 495.78,Z 454.73,A -85,B 0,C 180,E1 -6100.11,E2 -6100.11} C_VEL
LIN {X 0,Y 495.788,Z 454.727,A -85,B 0,C 180,E1 -6102.681,E2 -6102.681} C_VEL
LIN {X 0,Y 495.792,Z 454.727,A -85,B 0,C 180,E1 -6105.217,E2 -6105.217} C_VEL
LIN {X 0,Y 495.853,Z 454.717,A -85,B 0,C 180,E1 -6108.555,E2 -6108.555} C_VEL
LIN {X 0,Y 495.875,Z 454.717,A -85,B 0,C 180,E1 -6111.852,E2 -6111.852} C_VEL
LIN {X 0,Y 495.897,Z 454.714,A -85,B 0,C 180,E1 -6114.306,E2 -6114.306} C_VEL
LIN {X 0,Y 495.994,Z 454.702,A -85,B 0,C 180,E1 -6117.563,E2 -6117.563} C_VEL
LIN {X 0,Y 496,Z 454.704,A -85,B 0,C 180,E1 -6120,E2 -6120} C_VEL
LIN {X 0,Y 495.994,Z 454.7,A -85,B 0,C 180,E1 -6122.436,E2 -6122.436} C_VEL
LIN {X 0,Y 495.897,Z 454.714,A -85,B 0,C 180,E1 -6125.693,E2 -6125.693} C_VEL
LIN {X 0,Y 495.874,Z 454.718,A -85,B 0,C 180,E1 -6128.148,E2 -6128.148} C_VEL
LIN {X 0,Y 495.852,Z 454.721,A -85,B 0,C 180,E1 -6131.445,E2 -6131.445} C_VEL
LIN {X 0,Y 495.791,Z 454.727,A -85,B 0,C 180,E1 -6134.783,E2 -6134.783} C_VEL
LIN {X 0,Y 495.788,Z 454.73,A -85,B 0,C 180,E1 -6137.318,E2 -6137.318} C_VEL
LIN {X 0,Y 495.779,Z 454.728,A -85,B 0,C 180,E1 -6139.89,E2 -6139.89} C_VEL
LIN {X 0,Y 495.762,Z 454.73,A -85,B 0,C 180,E1 -6142.861,E2 -6142.861} C_VEL
LIN {X 0,Y 495.792,Z 454.726,A -85,B 0,C 180,E1 -6146.068,E2 -6146.068} C_VEL
LIN {X 0,Y 495.773,Z 454.73,A -85,B 0,C 180,E1 -6148.815,E2 -6148.815} C_VEL
LIN {X 0,Y 495.756,Z 454.732,A -85,B 0,C 180,E1 -6151.725,E2 -6151.725} C_VEL
LIN {X 0,Y 495.776,Z 454.732,A -85,B 0,C 180,E1 -6154.695,E2 -6154.695} C_VEL
LIN {X 0,Y 495.732,Z 454.738,A -85,B 0,C 180,E1 -6157.561,E2 -6157.561} C_VEL
LIN {X 0,Y 495.767,Z 454.732,A -85,B 0,C 180,E1 -6160.7,E2 -6160.7} C_VEL
LIN {X 0,Y 495.733,Z 454.737,A -85,B 0,C 180,E1 -6163.695,E2 -6163.695} C_VEL
LIN {X 0,Y 495.726,Z 454.738,A -85,B 0,C 180,E1 -6166.306,E2 -6166.306} C_VEL
LIN {X 0,Y 495.768,Z 454.732,A -85,B 0,C 180,E1 -6169.3,E2 -6169.3} C_VEL
LIN {X 0,Y 495.755,Z 454.778,A -85,B 0,C 180,E1 -6170.474,E2 -6170.474} C_VEL
LIN {X 0,Y 496.876,Z 460.955,A -85,B 0,C 180,E1 -6173.049,E2 -6173.049} C_VEL
LIN {X 0,Y 497.292,Z 464.83,A -85,B 0,C 180,E1 -6174.589,E2 -6174.589} C_VEL
LIN {X 0,Y 496.908,Z 472.576,A -85,B 0,C 180,E1 -6177.49,E2 -6177.49} C_VEL
LIN {X 0,Y 496.572,Z 480.354,A -85,B 0,C 180,E1 -6180.307,E2 -6180.307} C_VEL
LIN {X 0,Y 496.261,Z 488.455,A -85,B 0,C 180,E1 -6183.151,E2 -6183.151} C_VEL
LIN {X 0,Y 495.95,Z 497.359,A -85,B 0,C 180,E1 -6186.18,E2 -6186.18} C_VEL
LIN {X 0,Y 495.683,Z 506.577,A -85,B 0,C 180,E1 -6189.24,E2 -6189.24} C_VEL
LIN {X 0,Y 495.498,Z 515.896,A -85,B 0,C 180,E1 -6192.259,E2 -6192.259} C_VEL
LIN {X 0,Y 495.36,Z 525.145,A -85,B 0,C 180,E1 -6195.204,E2 -6195.204} C_VEL
LIN {X 0,Y 495.352,Z 526.043,A -85,B 0,C 180,E1 -6195.493,E2 -6195.493} C_VEL
LIN {X 0,Y 497.465,Z 540.564,A -85,B 0,C 180,E1 -6195.934,E2 -6195.934} C_VEL
LIN {X 0,Y 497.347,Z 552.85,A -85,B 0,C 180,E1 -6196.413,E2 -6196.413} C_VEL
LIN {X 0,Y 497.05,Z 564.49,A -85,B 0,C 180,E1 -6197.018,E2 -6197.018} C_VEL
LIN {X 0,Y 496.663,Z 575.457,A -85,B 0,C 180,E1 -6197.746,E2 -6197.746} C_VEL
LIN {X 0,Y 496.33,Z 585.444,A -85,B 0,C 180,E1 -6198.566,E2 -6198.566} C_VEL
LIN {X 0,Y 495.897,Z 595.54,A -85,B 0,C 180,E1 -6199.59,E2 -6199.59} C_VEL
LIN {X 0,Y 495.587,Z 605.32,A -85,B 0,C 180,E1 -6200.82,E2 -6200.82} C_VEL
LIN {X 0,Y 495.358,Z 613.136,A -85,B 0,C 180,E1 -6202.049,E2 -6202.049} C_VEL
LIN {X 0,Y 495.253,Z 618.476,A -85,B 0,C 180,E1 -6203.072,E2 -6203.072} C_VEL
LIN {X 0,Y 495.154,Z 623.657,A -85,B 0,C 180,E1 -6204.298,E2 -6204.298} C_VEL
LIN {X 0,Y 495.027,Z 627.67,A -85,B 0,C 180,E1 -6205.522,E2 -6205.522} C_VEL
LIN {X 0,Y 495.044,Z 630.636,A -85,B 0,C 180,E1 -6206.745,E2 -6206.745} C_VEL
LIN {X 0,Y 495.053,Z 632.049,A -85,B 0,C 180,E1 -6207.559,E2 -6207.559} C_VEL
LIN {X 0,Y 494.91,Z 633.653,A -85,B 0,C 180,E1 -6209.187,E2 -6209.187} C_VEL
LIN {X 0,Y 494.898,Z 633.862,A -85,B 0,C 180,E1 -6210,E2 -6210} C_VEL
LIN {X 0,Y 494.963,Z 633.014,A -85,B 0,C 180,E1 -6211.627,E2 -6211.627} C_VEL
LIN {X 0,Y 495.053,Z 631.995,A -85,B 0,C 180,E1 -6212.441,E2 -6212.441} C_VEL
LIN {X 0,Y 495.044,Z 630.558,A -85,B 0,C 180,E1 -6213.256,E2 -6213.256} C_VEL
LIN {X 0,Y 495.028,Z 627.551,A -85,B 0,C 180,E1 -6214.479,E2 -6214.479} C_VEL
LIN {X 0,Y 495.154,Z 623.49,A -85,B 0,C 180,E1 -6215.702,E2 -6215.702} C_VEL
LIN {X 0,Y 495.257,Z 617.238,A -85,B 0,C 180,E1 -6217.133,E2 -6217.133} C_VEL
LIN {X 0,Y 495.443,Z 610.41,A -85,B 0,C 180,E1 -6218.361,E2 -6218.361} C_VEL
LIN {X 0,Y 495.655,Z 601.926,A -85,B 0,C 180,E1 -6219.591,E2 -6219.591} C_VEL
LIN {X 0,Y 495.996,Z 593.215,A -85,B 0,C 180,E1 -6220.615,E2 -6220.615} C_VEL
LIN {X 0,Y 496.302,Z 582.483,A -85,B 0,C 180,E1 -6221.642,E2 -6221.642} C_VEL
LIN {X 0,Y 496.725,Z 571.214,A -85,B 0,C 180,E1 -6222.509,E2 -6222.509} C_VEL
LIN {X 0,Y 497.071,Z 560.222,A -85,B 0,C 180,E1 -6223.179,E2 -6223.179} C_VEL
LIN {X 0,Y 497.404,Z 546.962,A -85,B 0,C 180,E1 -6223.794,E2 -6223.794} C_VEL
LIN {X 0,Y 497.347,Z 540.228,A -85,B 0,C 180,E1 -6224.044,E2 -6224.044} C_VEL
LIN {X 0,Y 495.603,Z 527.755,A -85,B 0,C 180,E1 -6224.428,E2 -6224.428} C_VEL
LIN {X 0,Y 495.333,Z 525.173,A -85,B 0,C 180,E1 -6224.508,E2 -6224.508} C_VEL
LIN {X 0,Y 495.409,Z 515.995,A -85,B 0,C 180,E1 -6227.332,E2 -6227.332} C_VEL
LIN {X 0,Y 495.609,Z 505.5,A -85,B 0,C 180,E1 -6230.623,E2 -6230.623} C_VEL
LIN {X 0,Y 495.801,Z 495.614,A -85,B 0,C 180,E1 -6233.828,E2 -6233.828} C_VEL
LIN {X 0,Y 496.08,Z 486.42,A -85,B 0,C 180,E1 -6236.959,E2 -6236.959} C_VEL
LIN {X 0,Y 496.452,Z 477.352,A -85,B 0,C 180,E1 -6240.283,E2 -6240.283} C_VEL
LIN {X 0,Y 496.939,Z 469.517,A -85,B 0,C 180,E1 -6243.474,E2 -6243.474} C_VEL
LIN {X 0,Y 497.273,Z 465.304,A -85,B 0,C 180,E1 -6245.413,E2 -6245.413} C_VEL
LIN {X 0,Y 496.987,Z 461.529,A -85,B 0,C 180,E1 -6247.451,E2 -6247.451} C_VEL
LIN {X 0,Y 496.291,Z 457.693,A -85,B 0,C 180,E1 -6250.12,E2 -6250.12} C_VEL
LIN {X 0,Y 495.839,Z 455.296,A -85,B 0,C 180,E1 -6252.52,E2 -6252.52} C_VEL
LIN {X 0,Y 495.737,Z 454.737,A -85,B 0,C 180,E1 -6254.001,E2 -6254.001} C_VEL
LIN {X 0,Y 495.737,Z 454.737,A -85,B 0,C 180,E1 -6257.118,E2 -6257.118} C_VEL
LIN {X 0,Y 495.762,Z 454.734,A -85,B 0,C 180,E1 -6259.953,E2 -6259.953} C_VEL
LIN {X 0,Y 495.735,Z 454.847,A -85,B 0,C 180,E1 -6262.553,E2 -6262.553} C_VEL
LIN {X 0,Y 495.853,Z 456.446,A -85,B 0,C 180,E1 -6265.293,E2 -6265.293} C_VEL
LIN {X 0,Y 495.708,Z 458.673,A -85,B 0,C 180,E1 -6268.36,E2 -6268.36} C_VEL
LIN {X 0,Y 495.568,Z 461.244,A -85,B 0,C 180,E1 -6271.555,E2 -6271.555} C_VEL
LIN {X 0,Y 495.445,Z 463.296,A -85,B 0,C 180,E1 -6273.913,E2 -6273.913} C_VEL
LIN {X 0,Y 495.354,Z 465.717,A -85,B 0,C 180,E1 -6276.593,E2 -6276.593} C_VEL
LIN {X 0,Y 495.295,Z 468.43,A -85,B 0,C 180,E1 -6279.474,E2 -6279.474} C_VEL
LIN {X 0,Y 495.198,Z 471.563,A -85,B 0,C 180,E1 -6282.66,E2 -6282.66} C_VEL
LIN {X 0,Y 495.182,Z 474.603,A -85,B 0,C 180,E1 -6285.645,E2 -6285.645} C_VEL
LIN {X 0,Y 497.514,Z 486.029,A -85,B 0,C 180,E1 -6286.053,E2 -6286.053} C_VEL
LIN {X 0,Y 497.498,Z 497.507,A -85,B 0,C 180,E1 -6286.521,E2 -6286.521} C_VEL
LIN {X 0,Y 497.164,Z 509.405,A -85,B 0,C 180,E1 -6287.156,E2 -6287.156} C_VEL
LIN {X 0,Y 496.83,Z 520.969,A -85,B 0,C 180,E1 -6287.957,E2 -6287.957} C_VEL
LIN {X 0,Y 496.401,Z 531.549,A -85,B 0,C 180,E1 -6288.878,E2 -6288.878} C_VEL
LIN {X 0,Y 496.1,Z 540.2,A -85,B 0,C 180,E1 -6289.8,E2 -6289.8} C_VEL
LIN {X 0,Y 495.837,Z 548.154,A -85,B 0,C 180,E1 -6290.825,E2 -6290.825} C_VEL
LIN {X 0,Y 495.519,Z 555.948,A -85,B 0,C 180,E1 -6292.052,E2 -6292.052} C_VEL
LIN {X 0,Y 495.305,Z 562.419,A -85,B 0,C 180,E1 -6293.34,E2 -6293.34} C_VEL
LIN {X 0,Y 495.129,Z 567.772,A -85,B 0,C 180,E1 -6294.706,E2 -6294.706} C_VEL
LIN {X 0,Y 495.17,Z 571.38,A -85,B 0,C 180,E1 -6295.931,E2 -6295.931} C_VEL
LIN {X 0,Y 495.062,Z 573.246,A -85,B 0,C 180,E1 -6296.745,E2 -6296.745} C_VEL
LIN {X 0,Y 495.055,Z 574.654,A -85,B 0,C 180,E1 -6297.559,E2 -6297.559} C_VEL
LIN {X 0,Y 494.911,Z 576.258,A -85,B 0,C 180,E1 -6299.187,E2 -6299.187} C_VEL
LIN {X 0,Y 494.9,Z 576.482,A -85,B 0,C 180,E1 -6300,E2 -6300} C_VEL
LIN {X 0,Y 494.911,Z 576.285,A -85,B 0,C 180,E1 -6300.814,E2 -6300.814} C_VEL
LIN {X 0,Y 495.054,Z 574.695,A -85,B 0,C 180,E1 -6302.441,E2 -6302.441} C_VEL
LIN {X 0,Y 495.051,Z 573.319,A -85,B 0,C 180,E1 -6303.256,E2 -6303.256} C_VEL
LIN {X 0,Y 495.138,Z 570.417,A -85,B 0,C 180,E1 -6304.478,E2 -6304.478} C_VEL
LIN {X 0,Y 495.229,Z 566.487,A -85,B 0,C 180,E1 -6305.701,E2 -6305.701} C_VEL
LIN {X 0,Y 495.358,Z 561.421,A -85,B 0,C 180,E1 -6306.926,E2 -6306.926} C_VEL
LIN {X 0,Y 495.515,Z 555.029,A -85,B 0,C 180,E1 -6308.154,E2 -6308.154} C_VEL
LIN {X 0,Y 495.762,Z 547.044,A -85,B 0,C 180,E1 -6309.383,E2 -6309.383} C_VEL
LIN {X 0,Y 496.113,Z 538.896,A -85,B 0,C 180,E1 -6310.406,E2 -6310.406} C_VEL
LIN {X 0,Y 496.508,Z 528.962,A -85,B 0,C 180,E1 -6311.43,E2 -6311.43} C_VEL
LIN {X 0,Y 496.87,Z 518.151,A -85,B 0,C 180,E1 -6312.323,E2 -6312.323} C_VEL
LIN {X 0,Y 497.173,Z 506.78,A -85,B 0,C 180,E1 -6313.072,E2 -6313.072} C_VEL
LIN {X 0,Y 497.539,Z 494.706,A -85,B 0,C 180,E1 -6313.686,E2 -6313.686} C_VEL
LIN {X 0,Y 497.542,Z 486.464,A -85,B 0,C 180,E1 -6314.012,E2 -6314.012} C_VEL
LIN {X 0,Y 495.668,Z 476.279,A -85,B 0,C 180,E1 -6314.376,E2 -6314.376} C_VEL
LIN {X 0,Y 495.086,Z 473.507,A -85,B 0,C 180,E1 -6314.473,E2 -6314.473} C_VEL
LIN {X 0,Y 495.101,Z 469.55,A -85,B 0,C 180,E1 -6317.996,E2 -6317.996} C_VEL
LIN {X 0,Y 495.096,Z 466.462,A -85,B 0,C 180,E1 -6320.786,E2 -6320.786} C_VEL
LIN {X 0,Y 495.14,Z 463.562,A -85,B 0,C 180,E1 -6323.418,E2 -6323.418} C_VEL
LIN {X 0,Y 495.239,Z 460.102,A -85,B 0,C 180,E1 -6326.614,E2 -6326.614} C_VEL
LIN {X 0,Y 495.278,Z 456.402,A -85,B 0,C 180,E1 -6330.049,E2 -6330.049} C_VEL
LIN {X 0,Y 495.268,Z 454.796,A -85,B 0,C 180,E1 -6331.671,E2 -6331.671} C_VEL
LIN {X 0,Y 495.63,Z 454.75,A -85,B 0,C 180,E1 -6334.67,E2 -6334.67} C_VEL
LIN {X 0,Y 495.724,Z 454.734,A -85,B 0,C 180,E1 -6337.563,E2 -6337.563} C_VEL
LIN {X 0,Y 495.764,Z 454.734,A -85,B 0,C 180,E1 -6340.047,E2 -6340.047} C_VEL
LIN {X 0,Y 495.731,Z 454.737,A -85,B 0,C 180,E1 -6342.883,E2 -6342.883} C_VEL
LIN {X 0,Y 495.732,Z 454.736,A -85,B 0,C 180,E1 -6345.998,E2 -6345.998} C_VEL
LIN {X 0,Y 495.771,Z 454.731,A -85,B 0,C 180,E1 -6349.3,E2 -6349.3} C_VEL
LIN {X 0,Y 495.735,Z 454.737,A -85,B 0,C 180,E1 -6352.439,E2 -6352.439} C_VEL
LIN {X 0,Y 495.784,Z 454.73,A -85,B 0,C 180,E1 -6355.457,E2 -6355.457} C_VEL
LIN {X 0,Y 495.797,Z 454.728,A -85,B 0,C 180,E1 -6356.767,E2 -6356.767} C_VEL
LIN {X 0,Y 495.093,Z 454.815,A -85,B 0,C 180,E1 -6357.444,E2 -6357.444} C_VEL
LIN {X 0,Y 492.215,Z 455.176,A -85,B 0,C 180,E1 -6358.544,E2 -6358.544} C_VEL
LIN {X 0,Y 489.81,Z 455.472,A -85,B 0,C 180,E1 -6359.431,E2 -6359.431} C_VEL
LIN {X 0,Y 488.79,Z 455.602,A -85,B 0,C 180,E1 -6360.116,E2 -6360.116} C_VEL
LIN {X 0,Y 488.712,Z 455.606,A -85,B 0,C 180,E1 -6360.347,E2 -6360.347} C_VEL
LIN {X 0,Y 488.763,Z 455.605,A -85,B 0,C 180,E1 -6363.528,E2 -6363.528} C_VEL
LIN {X 0,Y 488.696,Z 455.614,A -85,B 0,C 180,E1 -6366.254,E2 -6366.254} C_VEL
LIN {X 0,Y 488.752,Z 455.604,A -85,B 0,C 180,E1 -6369.176,E2 -6369.176} C_VEL
LIN {X 0,Y 488.766,Z 455.603,A -85,B 0,C 180,E1 -6371.628,E2 -6371.628} C_VEL
LIN {X 0,Y 488.768,Z 455.6,A -85,B 0,C 180,E1 -6375,E2 -6375} C_VEL
LIN {X 0,Y 488.812,Z 455.597,A -85,B 0,C 180,E1 -6378.388,E2 -6378.388} C_VEL
LIN {X 0,Y 488.791,Z 455.6,A -85,B 0,C 180,E1 -6381.733,E2 -6381.733} C_VEL
LIN {X 0,Y 488.86,Z 455.59,A -85,B 0,C 180,E1 -6384.224,E2 -6384.224} C_VEL
LIN {X 0,Y 488.966,Z 455.576,A -85,B 0,C 180,E1 -6387.528,E2 -6387.528} C_VEL
LIN {X 0,Y 488.961,Z 455.577,A -85,B 0,C 180,E1 -6390.823,E2 -6390.823} C_VEL
LIN {X 0,Y 488.966,Z 455.578,A -85,B 0,C 180,E1 -6392.471,E2 -6392.471} C_VEL
LIN {X 0,Y 488.844,Z 455.594,A -85,B 0,C 180,E1 -6395.776,E2 -6395.776} C_VEL
LIN {X 0,Y 488.823,Z 455.595,A -85,B 0,C 180,E1 -6398.266,E2 -6398.266} C_VEL
LIN {X 0,Y 488.812,Z 455.596,A -85,B 0,C 180,E1 -6401.612,E2 -6401.612} C_VEL
LIN {X 0,Y 488.768,Z 455.602,A -85,B 0,C 180,E1 -6405,E2 -6405} C_VEL
LIN {X 0,Y 488.76,Z 455.605,A -85,B 0,C 180,E1 -6408.442,E2 -6408.442} C_VEL
LIN {X 0,Y 488.712,Z 455.607,A -85,B 0,C 180,E1 -6411.07,E2 -6411.07} C_VEL
LIN {X 0,Y 488.694,Z 455.612,A -85,B 0,C 180,E1 -6413.745,E2 -6413.745} C_VEL
LIN {X 0,Y 488.796,Z 455.597,A -85,B 0,C 180,E1 -6416.943,E2 -6416.943} C_VEL
LIN {X 0,Y 488.714,Z 455.608,A -85,B 0,C 180,E1 -6420.362,E2 -6420.362} C_VEL
LIN {X 0,Y 488.74,Z 455.605,A -85,B 0,C 180,E1 -6423.484,E2 -6423.484} C_VEL
LIN {X 0,Y 488.691,Z 455.61,A -85,B 0,C 180,E1 -6426.355,E2 -6426.355} C_VEL
LIN {X 0,Y 488.704,Z 455.611,A -85,B 0,C 180,E1 -6429.254,E2 -6429.254} C_VEL
LIN {X 0,Y 488.71,Z 455.61,A -85,B 0,C 180,E1 -6431.599,E2 -6431.599} C_VEL
LIN {X 0,Y 488.715,Z 455.609,A -85,B 0,C 180,E1 -6434.801,E2 -6434.801} C_VEL
LIN {X 0,Y 488.698,Z 455.61,A -85,B 0,C 180,E1 -6437.475,E2 -6437.475} C_VEL
LIN {X 0,Y 488.735,Z 455.609,A -85,B 0,C 180,E1 -6439.676,E2 -6439.676} C_VEL
LIN {X 0,Y 488.685,Z 455.614,A -85,B 0,C 180,E1 -6442.841,E2 -6442.841} C_VEL
LIN {X 0,Y 488.737,Z 455.61,A -85,B 0,C 180,E1 -6445.887,E2 -6445.887} C_VEL
LIN {X 0,Y 488.695,Z 455.612,A -85,B 0,C 180,E1 -6448.82,E2 -6448.82} C_VEL
LIN {X 0,Y 488.747,Z 455.605,A -85,B 0,C 180,E1 -6451.671,E2 -6451.671} C_VEL
LIN {X 0,Y 488.749,Z 455.602,A -85,B 0,C 180,E1 -6454.444,E2 -6454.444} C_VEL
LIN {X 0,Y 488.725,Z 455.61,A -85,B 0,C 180,E1 -6457.153,E2 -6457.153} C_VEL
LIN {X 0,Y 488.731,Z 455.61,A -85,B 0,C 180,E1 -6459.81,E2 -6459.81} C_VEL
LIN {X 0,Y 488.736,Z 455.605,A -85,B 0,C 180,E1 -6462.423,E2 -6462.423} C_VEL
LIN {X 0,Y 488.764,Z 455.604,A -85,B 0,C 180,E1 -6464.999,E2 -6464.999} C_VEL
LIN {X 0,Y 488.807,Z 455.595,A -85,B 0,C 180,E1 -6468.387,E2 -6468.387} C_VEL
LIN {X 0,Y 488.819,Z 455.596,A -85,B 0,C 180,E1 -6471.733,E2 -6471.733} C_VEL
LIN {X 0,Y 488.856,Z 455.591,A -85,B 0,C 180,E1 -6474.224,E2 -6474.224} C_VEL
LIN {X 0,Y 488.962,Z 455.579,A -85,B 0,C 180,E1 -6477.528,E2 -6477.528} C_VEL
LIN {X 0,Y 488.956,Z 455.578,A -85,B 0,C 180,E1 -6480.823,E2 -6480.823} C_VEL
LIN {X 0,Y 488.962,Z 455.576,A -85,B 0,C 180,E1 -6482.471,E2 -6482.471} C_VEL
LIN {X 0,Y 488.856,Z 455.591,A -85,B 0,C 180,E1 -6485.776,E2 -6485.776} C_VEL
LIN {X 0,Y 488.818,Z 455.596,A -85,B 0,C 180,E1 -6488.266,E2 -6488.266} C_VEL
LIN {X 0,Y 488.806,Z 455.598,A -85,B 0,C 180,E1 -6491.612,E2 -6491.612} C_VEL
LIN {X 0,Y 488.763,Z 455.602,A -85,B 0,C 180,E1 -6495,E2 -6495} C_VEL
LIN {X 0,Y 488.756,Z 455.602,A -85,B 0,C 180,E1 -6498.442,E2 -6498.442} C_VEL
LIN {X 0,Y 488.708,Z 455.61,A -85,B 0,C 180,E1 -6501.071,E2 -6501.071} C_VEL
LIN {X 0,Y 488.694,Z 455.613,A -85,B 0,C 180,E1 -6503.745,E2 -6503.745} C_VEL
LIN {X 0,Y 488.793,Z 455.602,A -85,B 0,C 180,E1 -6506.944,E2 -6506.944} C_VEL
LIN {X 0,Y 488.71,Z 455.609,A -85,B 0,C 180,E1 -6510.363,E2 -6510.363} C_VEL
LIN {X 0,Y 488.736,Z 455.606,A -85,B 0,C 180,E1 -6513.484,E2 -6513.484} C_VEL
LIN {X 0,Y 488.689,Z 455.613,A -85,B 0,C 180,E1 -6516.356,E2 -6516.356} C_VEL
LIN {X 0,Y 488.701,Z 455.614,A -85,B 0,C 180,E1 -6519.254,E2 -6519.254} C_VEL
LIN {X 0,Y 488.736,Z 455.608,A -85,B 0,C 180,E1 -6522.521,E2 -6522.521} C_VEL
LIN {X 0,Y 488.694,Z 455.615,A -85,B 0,C 180,E1 -6525.977,E2 -6525.977} C_VEL
LIN {X 0,Y 488.709,Z 455.614,A -85,B 0,C 180,E1 -6528.585,E2 -6528.585} C_VEL
LIN {X 0,Y 488.734,Z 455.654,A -85,B 0,C 180,E1 -6530.215,E2 -6530.215} C_VEL
LIN {X 0,Y 490.076,Z 463.268,A -85,B 0,C 180,E1 -6533.425,E2 -6533.425} C_VEL
LIN {X 0,Y 490.241,Z 467.269,A -85,B 0,C 180,E1 -6535.01,E2 -6535.01} C_VEL
LIN {X 0,Y 489.865,Z 475.018,A -85,B 0,C 180,E1 -6537.938,E2 -6537.938} C_VEL
LIN {X 0,Y 489.433,Z 483.836,A -85,B 0,C 180,E1 -6541.155,E2 -6541.155} C_VEL
LIN {X 0,Y 489.128,Z 491.91,A -85,B 0,C 180,E1 -6544.009,E2 -6544.009} C_VEL
LIN {X 0,Y 488.812,Z 500.47,A -85,B 0,C 180,E1 -6546.952,E2 -6546.952} C_VEL
LIN {X 0,Y 488.6,Z 508.983,A -85,B 0,C 180,E1 -6549.805,E2 -6549.805} C_VEL
LIN {X 0,Y 488.406,Z 518.214,A -85,B 0,C 180,E1 -6552.843,E2 -6552.843} C_VEL
LIN {X 0,Y 488.287,Z 525.721,A -85,B 0,C 180,E1 -6555.278,E2 -6555.278} C_VEL
LIN {X 0,Y 490.485,Z 541.157,A -85,B 0,C 180,E1 -6555.769,E2 -6555.769} C_VEL
LIN {X 0,Y 490.491,Z 551.178,A -85,B 0,C 180,E1 -6556.166,E2 -6556.166} C_VEL
LIN {X 0,Y 490.138,Z 562.378,A -85,B 0,C 180,E1 -6556.737,E2 -6556.737} C_VEL
LIN {X 0,Y 489.673,Z 574.939,A -85,B 0,C 180,E1 -6557.568,E2 -6557.568} C_VEL
LIN {X 0,Y 489.297,Z 586.049,A -85,B 0,C 180,E1 -6558.505,E2 -6558.505} C_VEL
LIN {X 0,Y 488.821,Z 596.859,A -85,B 0,C 180,E1 -6559.647,E2 -6559.647} C_VEL
LIN {X 0,Y 488.518,Z 604.859,A -85,B 0,C 180,E1 -6560.686,E2 -6560.686} C_VEL
LIN {X 0,Y 488.291,Z 612.696,A -85,B 0,C 180,E1 -6561.933,E2 -6561.933} C_VEL
LIN {X 0,Y 488.069,Z 619.886,A -85,B 0,C 180,E1 -6563.385,E2 -6563.385} C_VEL
LIN {X 0,Y 488.052,Z 624.683,A -85,B 0,C 180,E1 -6564.629,E2 -6564.629} C_VEL
LIN {X 0,Y 487.958,Z 628.34,A -85,B 0,C 180,E1 -6565.87,E2 -6565.87} C_VEL
LIN {X 0,Y 487.968,Z 630.229,A -85,B 0,C 180,E1 -6566.698,E2 -6566.698} C_VEL
LIN {X 0,Y 487.959,Z 631.643,A -85,B 0,C 180,E1 -6567.524,E2 -6567.524} C_VEL
LIN {X 0,Y 487.893,Z 632.644,A -85,B 0,C 180,E1 -6568.349,E2 -6568.349} C_VEL
LIN {X 0,Y 487.819,Z 633.453,A -85,B 0,C 180,E1 -6570,E2 -6570} C_VEL
LIN {X 0,Y 487.893,Z 632.597,A -85,B 0,C 180,E1 -6571.651,E2 -6571.651} C_VEL
LIN {X 0,Y 487.972,Z 631.567,A -85,B 0,C 180,E1 -6572.477,E2 -6572.477} C_VEL
LIN {X 0,Y 487.969,Z 630.121,A -85,B 0,C 180,E1 -6573.303,E2 -6573.303} C_VEL
LIN {X 0,Y 487.937,Z 627.097,A -85,B 0,C 180,E1 -6574.544,E2 -6574.544} C_VEL
LIN {X 0,Y 488.05,Z 623.014,A -85,B 0,C 180,E1 -6575.785,E2 -6575.785} C_VEL
LIN {X 0,Y 488.183,Z 616.734,A -85,B 0,C 180,E1 -6577.237,E2 -6577.237} C_VEL
LIN {X 0,Y 488.369,Z 609.869,A -85,B 0,C 180,E1 -6578.483,E2 -6578.483} C_VEL
LIN {X 0,Y 488.601,Z 601.351,A -85,B 0,C 180,E1 -6579.731,E2 -6579.731} C_VEL
LIN {X 0,Y 488.949,Z 592.599,A -85,B 0,C 180,E1 -6580.77,E2 -6580.77} C_VEL
LIN {X 0,Y 489.307,Z 581.83,A -85,B 0,C 180,E1 -6581.811,E2 -6581.811} C_VEL
LIN {X 0,Y 489.735,Z 570.331,A -85,B 0,C 180,E1 -6582.703,E2 -6582.703} C_VEL
LIN {X 0,Y 490.105,Z 559.468,A -85,B 0,C 180,E1 -6583.37,E2 -6583.37} C_VEL
LIN {X 0,Y 490.513,Z 546.202,A -85,B 0,C 180,E1 -6583.992,E2 -6583.992} C_VEL
LIN {X 0,Y 490.358,Z 540.549,A -85,B 0,C 180,E1 -6584.208,E2 -6584.208} C_VEL
LIN {X 0,Y 488.519,Z 527.247,A -85,B 0,C 180,E1 -6584.635,E2 -6584.635} C_VEL
LIN {X 0,Y 488.24,Z 524.739,A -85,B 0,C 180,E1 -6584.697,E2 -6584.697} C_VEL
LIN {X 0,Y 488.317,Z 515.513,A -85,B 0,C 180,E1 -6587.592,E2 -6587.592} C_VEL
LIN {X 0,Y 488.542,Z 505.628,A -85,B 0,C 180,E1 -6590.761,E2 -6590.761} C_VEL
LIN {X 0,Y 488.738,Z 496.62,A -85,B 0,C 180,E1 -6593.743,E2 -6593.743} C_VEL
LIN {X 0,Y 489.05,Z 487.256,A -85,B 0,C 180,E1 -6597.003,E2 -6597.003} C_VEL
LIN {X 0,Y 489.394,Z 478.773,A -85,B 0,C 180,E1 -6600.174,E2 -6600.174} C_VEL
LIN {X 0,Y 489.855,Z 471.837,A -85,B 0,C 180,E1 -6603.038,E2 -6603.038} C_VEL
LIN {X 0,Y 490.28,Z 467.136,A -85,B 0,C 180,E1 -6605.207,E2 -6605.207} C_VEL
LIN {X 0,Y 490.125,Z 463.758,A -85,B 0,C 180,E1 -6607.031,E2 -6607.031} C_VEL
LIN {X 0,Y 489.602,Z 460.473,A -85,B 0,C 180,E1 -6609.182,E2 -6609.182} C_VEL
LIN {X 0,Y 489.069,Z 457.644,A -85,B 0,C 180,E1 -6611.647,E2 -6611.647} C_VEL
LIN {X 0,Y 488.735,Z 455.881,A -85,B 0,C 180,E1 -6614.028,E2 -6614.028} C_VEL
LIN {X 0,Y 488.696,Z 455.614,A -85,B 0,C 180,E1 -6616.346,E2 -6616.346} C_VEL
LIN {X 0,Y 488.722,Z 455.611,A -85,B 0,C 180,E1 -6618.586,E2 -6618.586} C_VEL
LIN {X 0,Y 488.712,Z 455.794,A -85,B 0,C 180,E1 -6621.803,E2 -6621.803} C_VEL
LIN {X 0,Y 488.841,Z 456.779,A -85,B 0,C 180,E1 -6623.882,E2 -6623.882} C_VEL
LIN {X 0,Y 488.766,Z 458.661,A -85,B 0,C 180,E1 -6626.879,E2 -6626.879} C_VEL
LIN {X 0,Y 488.624,Z 460.804,A -85,B 0,C 180,E1 -6629.774,E2 -6629.774} C_VEL
LIN {X 0,Y 488.475,Z 463.082,A -85,B 0,C 180,E1 -6632.587,E2 -6632.587} C_VEL
LIN {X 0,Y 488.382,Z 465.456,A -85,B 0,C 180,E1 -6635.334,E2 -6635.334} C_VEL
LIN {X 0,Y 488.245,Z 467.905,A -85,B 0,C 180,E1 -6638.022,E2 -6638.022} C_VEL
LIN {X 0,Y 488.154,Z 470.399,A -85,B 0,C 180,E1 -6640.662,E2 -6640.662} C_VEL
LIN {X 0,Y 488.139,Z 472.939,A -85,B 0,C 180,E1 -6643.265,E2 -6643.265} C_VEL
LIN {X 0,Y 488.17,Z 475.331,A -85,B 0,C 180,E1 -6645.449,E2 -6645.449} C_VEL
LIN {X 0,Y 490.613,Z 486.669,A -85,B 0,C 180,E1 -6645.866,E2 -6645.866} C_VEL
LIN {X 0,Y 490.631,Z 496.663,A -85,B 0,C 180,E1 -6646.276,E2 -6646.276} C_VEL
LIN {X 0,Y 490.238,Z 509.882,A -85,B 0,C 180,E1 -6646.986,E2 -6646.986} C_VEL
LIN {X 0,Y 489.906,Z 521.254,A -85,B 0,C 180,E1 -6647.784,E2 -6647.784} C_VEL
LIN {X 0,Y 489.451,Z 531.856,A -85,B 0,C 180,E1 -6648.718,E2 -6648.718} C_VEL
LIN {X 0,Y 489.119,Z 540.531,A -85,B 0,C 180,E1 -6649.653,E2 -6649.653} C_VEL
LIN {X 0,Y 488.836,Z 548.506,A -85,B 0,C 180,E1 -6650.692,E2 -6650.692} C_VEL
LIN {X 0,Y 488.505,Z 556.323,A -85,B 0,C 180,E1 -6651.937,E2 -6651.937} C_VEL
LIN {X 0,Y 488.265,Z 563.073,A -85,B 0,C 180,E1 -6653.304,E2 -6653.304} C_VEL
LIN {X 0,Y 488.074,Z 568.177,A -85,B 0,C 180,E1 -6654.63,E2 -6654.63} C_VEL
LIN {X 0,Y 488.106,Z 571.792,A -85,B 0,C 180,E1 -6655.872,E2 -6655.872} C_VEL
LIN {X 0,Y 487.99,Z 573.661,A -85,B 0,C 180,E1 -6656.698,E2 -6656.698} C_VEL
LIN {X 0,Y 487.991,Z 575.071,A -85,B 0,C 180,E1 -6657.524,E2 -6657.524} C_VEL
LIN {X 0,Y 487.834,Z 576.672,A -85,B 0,C 180,E1 -6659.175,E2 -6659.175} C_VEL
LIN {X 0,Y 487.82,Z 576.895,A -85,B 0,C 180,E1 -6660,E2 -6660} C_VEL
LIN {X 0,Y 487.834,Z 576.692,A -85,B 0,C 180,E1 -6660.826,E2 -6660.826} C_VEL
LIN {X 0,Y 487.989,Z 575.087,A -85,B 0,C 180,E1 -6662.476,E2 -6662.476} C_VEL
LIN {X 0,Y 487.98,Z 573.705,A -85,B 0,C 180,E1 -6663.303,E2 -6663.303} C_VEL
LIN {X 0,Y 488.069,Z 570.789,A -85,B 0,C 180,E1 -6664.543,E2 -6664.543} C_VEL
LIN {X 0,Y 488.179,Z 566.841,A -85,B 0,C 180,E1 -6665.784,E2 -6665.784} C_VEL
LIN {X 0,Y 488.336,Z 560.859,A -85,B 0,C 180,E1 -6667.214,E2 -6667.214} C_VEL
LIN {X 0,Y 488.551,Z 554.101,A -85,B 0,C 180,E1 -6668.479,E2 -6668.479} C_VEL
LIN {X 0,Y 488.841,Z 545.836,A -85,B 0,C 180,E1 -6669.726,E2 -6669.726} C_VEL
LIN {X 0,Y 489.152,Z 537.348,A -85,B 0,C 180,E1 -6670.765,E2 -6670.765} C_VEL
LIN {X 0,Y 489.664,Z 526.865,A -85,B 0,C 180,E1 -6671.802,E2 -6671.802} C_VEL
LIN {X 0,Y 489.97,Z 516.118,A -85,B 0,C 180,E1 -6672.665,E2 -6672.665} C_VEL
LIN {X 0,Y 490.307,Z 505.19,A -85,B 0,C 180,E1 -6673.364,E2 -6673.364} C_VEL
LIN {X 0,Y 490.7,Z 492.329,A -85,B 0,C 180,E1 -6673.987,E2 -6673.987} C_VEL
LIN {X 0,Y 490.559,Z 486.559,A -85,B 0,C 180,E1 -6674.216,E2 -6674.216} C_VEL
LIN {X 0,Y 488.41,Z 475.817,A -85,B 0,C 180,E1 -6674.607,E2 -6674.607} C_VEL
LIN {X 0,Y 488.018,Z 473.84,A -85,B 0,C 180,E1 -6674.677,E2 -6674.677} C_VEL
LIN {X 0,Y 488.036,Z 469.992,A -85,B 0,C 180,E1 -6678.113,E2 -6678.113} C_VEL
LIN {X 0,Y 488.014,Z 466.694,A -85,B 0,C 180,E1 -6681.102,E2 -6681.102} C_VEL
LIN {X 0,Y 488.066,Z 463.778,A -85,B 0,C 180,E1 -6683.778,E2 -6683.778} C_VEL
LIN {X 0,Y 488.173,Z 460.512,A -85,B 0,C 180,E1 -6686.799,E2 -6686.799} C_VEL
LIN {X 0,Y 488.219,Z 456.831,A -85,B 0,C 180,E1 -6690.254,E2 -6690.254} C_VEL
LIN {X 0,Y 488.178,Z 455.819,A -85,B 0,C 180,E1 -6691.217,E2 -6691.217} C_VEL
LIN {X 0,Y 488.522,Z 455.636,A -85,B 0,C 180,E1 -6694.13,E2 -6694.13} C_VEL
LIN {X 0,Y 488.671,Z 455.614,A -85,B 0,C 180,E1 -6697.16,E2 -6697.16} C_VEL
LIN {X 0,Y 488.723,Z 455.608,A -85,B 0,C 180,E1 -6700.345,E2 -6700.345} C_VEL
LIN {X 0,Y 488.69,Z 455.611,A -85,B 0,C 180,E1 -6703.655,E2 -6703.655} C_VEL
LIN {X 0,Y 488.689,Z 455.614,A -85,B 0,C 180,E1 -6706.345,E2 -6706.345} C_VEL
LIN {X 0,Y 488.738,Z 455.607,A -85,B 0,C 180,E1 -6709.677,E2 -6709.677} C_VEL
LIN {X 0,Y 488.685,Z 455.611,A -85,B 0,C 180,E1 -6712.841,E2 -6712.841} C_VEL
LIN {X 0,Y 488.736,Z 455.607,A -85,B 0,C 180,E1 -6715.887,E2 -6715.887} C_VEL
LIN {X 0,Y 488.697,Z 455.611,A -85,B 0,C 180,E1 -6718.82,E2 -6718.82} C_VEL
LIN {X 0,Y 488.712,Z 455.606,A -85,B 0,C 180,E1 -6720.347,E2 -6720.347} C_VEL
LIN {X 0,Y 488.059,Z 455.689,A -85,B 0,C 180,E1 -6721.036,E2 -6721.036} C_VEL
LIN {X 0,Y 485.215,Z 456.046,A -85,B 0,C 180,E1 -6722.154,E2 -6722.154} C_VEL
LIN {X 0,Y 482.809,Z 456.345,A -85,B 0,C 180,E1 -6723.055,E2 -6723.055} C_VEL
LIN {X 0,Y 481.784,Z 456.473,A -85,B 0,C 180,E1 -6723.751,E2 -6723.751} C_VEL
LIN {X 0,Y 481.706,Z 456.481,A -85,B 0,C 180,E1 -6723.987,E2 -6723.987} C_VEL
LIN {X 0,Y 481.68,Z 456.484,A -85,B 0,C 180,E1 -6726.812,E2 -6726.812} C_VEL
LIN {X 0,Y 481.702,Z 456.484,A -85,B 0,C 180,E1 -6729.503,E2 -6729.503} C_VEL
LIN {X 0,Y 481.71,Z 456.482,A -85,B 0,C 180,E1 -6732.158,E2 -6732.158} C_VEL
LIN {X 0,Y 481.749,Z 456.475,A -85,B 0,C 180,E1 -6734.776,E2 -6734.776} C_VEL
LIN {X 0,Y 481.757,Z 456.475,A -85,B 0,C 180,E1 -6738.215,E2 -6738.215} C_VEL
LIN {X 0,Y 481.746,Z 456.476,A -85,B 0,C 180,E1 -6741.611,E2 -6741.611} C_VEL
LIN {X 0,Y 481.821,Z 456.468,A -85,B 0,C 180,E1 -6744.139,E2 -6744.139} C_VEL
LIN {X 0,Y 481.933,Z 456.453,A -85,B 0,C 180,E1 -6747.492,E2 -6747.492} C_VEL
LIN {X 0,Y 481.912,Z 456.456,A -85,B 0,C 180,E1 -6750.835,E2 -6750.835} C_VEL
LIN {X 0,Y 481.933,Z 456.454,A -85,B 0,C 180,E1 -6752.507,E2 -6752.507} C_VEL
LIN {X 0,Y 481.803,Z 456.471,A -85,B 0,C 180,E1 -6755.86,E2 -6755.86} C_VEL
LIN {X 0,Y 481.769,Z 456.473,A -85,B 0,C 180,E1 -6758.388,E2 -6758.388} C_VEL
LIN {X 0,Y 481.757,Z 456.476,A -85,B 0,C 180,E1 -6761.785,E2 -6761.785} C_VEL
LIN {X 0,Y 481.748,Z 456.477,A -85,B 0,C 180,E1 -6765.224,E2 -6765.224} C_VEL
LIN {X 0,Y 481.717,Z 456.481,A -85,B 0,C 180,E1 -6768.721,E2 -6768.721} C_VEL
LIN {X 0,Y 481.651,Z 456.488,A -85,B 0,C 180,E1 -6771.394,E2 -6771.394} C_VEL
LIN {X 0,Y 481.679,Z 456.485,A -85,B 0,C 180,E1 -6774.113,E2 -6774.113} C_VEL
LIN {X 0,Y 481.751,Z 456.475,A -85,B 0,C 180,E1 -6777.139,E2 -6777.139} C_VEL
LIN {X 0,Y 481.683,Z 456.486,A -85,B 0,C 180,E1 -6779.741,E2 -6779.741} C_VEL
LIN {X 0,Y 481.676,Z 456.486,A -85,B 0,C 180,E1 -6782.674,E2 -6782.674} C_VEL
LIN {X 0,Y 481.645,Z 456.493,A -85,B 0,C 180,E1 -6785.709,E2 -6785.709} C_VEL
LIN {X 0,Y 481.674,Z 456.487,A -85,B 0,C 180,E1 -6788.859,E2 -6788.859} C_VEL
LIN {X 0,Y 481.655,Z 456.491,A -85,B 0,C 180,E1 -6791.912,E2 -6791.912} C_VEL
LIN {X 0,Y 481.663,Z 456.487,A -85,B 0,C 180,E1 -6794.457,E2 -6794.457} C_VEL
LIN {X 0,Y 481.657,Z 456.489,A -85,B 0,C 180,E1 -6797.84,E2 -6797.84} C_VEL
LIN {X 0,Y 481.664,Z 456.486,A -85,B 0,C 180,E1 -6800.654,E2 -6800.654} C_VEL
LIN {X 0,Y 481.634,Z 456.491,A -85,B 0,C 180,E1 -6803.375,E2 -6803.375} C_VEL
LIN {X 0,Y 481.712,Z 456.48,A -85,B 0,C 180,E1 -6806.33,E2 -6806.33} C_VEL
LIN {X 0,Y 481.653,Z 456.49,A -85,B 0,C 180,E1 -6809.417,E2 -6809.417} C_VEL
LIN {X 0,Y 481.703,Z 456.484,A -85,B 0,C 180,E1 -6812.168,E2 -6812.168} C_VEL
LIN {X 0,Y 481.719,Z 456.479,A -85,B 0,C 180,E1 -6814.97,E2 -6814.97} C_VEL
LIN {X 0,Y 481.651,Z 456.489,A -85,B 0,C 180,E1 -6817.704,E2 -6817.704} C_VEL
LIN {X 0,Y 481.71,Z 456.48,A -85,B 0,C 180,E1 -6820.393,E2 -6820.393} C_VEL
LIN {X 0,Y 481.693,Z 456.485,A -85,B 0,C 180,E1 -6823.034,E2 -6823.034} C_VEL
LIN {X 0,Y 481.691,Z 456.484,A -85,B 0,C 180,E1 -6825.638,E2 -6825.638} C_VEL
LIN {X 0,Y 481.752,Z 456.474,A -85,B 0,C 180,E1 -6828.215,E2 -6828.215} C_VEL
LIN {X 0,Y 481.765,Z 456.474,A -85,B 0,C 180,E1 -6831.611,E2 -6831.611} C_VEL
LIN {X 0,Y 481.817,Z 456.469,A -85,B 0,C 180,E1 -6834.139,E2 -6834.139} C_VEL
LIN {X 0,Y 481.929,Z 456.455,A -85,B 0,C 180,E1 -6837.492,E2 -6837.492} C_VEL
LIN {X 0,Y 481.907,Z 456.456,A -85,B 0,C 180,E1 -6840.835,E2 -6840.835} C_VEL
LIN {X 0,Y 481.928,Z 456.452,A -85,B 0,C 180,E1 -6842.507,E2 -6842.507} C_VEL
LIN {X 0,Y 481.817,Z 456.468,A -85,B 0,C 180,E1 -6845.86,E2 -6845.86} C_VEL
LIN {X 0,Y 481.763,Z 456.475,A -85,B 0,C 180,E1 -6848.388,E2 -6848.388} C_VEL
LIN {X 0,Y 481.752,Z 456.476,A -85,B 0,C 180,E1 -6851.785,E2 -6851.785} C_VEL
LIN {X 0,Y 481.744,Z 456.477,A -85,B 0,C 180,E1 -6855.224,E2 -6855.224} C_VEL
LIN {X 0,Y 481.713,Z 456.481,A -85,B 0,C 180,E1 -6858.722,E2 -6858.722} C_VEL
LIN {X 0,Y 481.646,Z 456.489,A -85,B 0,C 180,E1 -6861.395,E2 -6861.395} C_VEL
LIN {X 0,Y 481.678,Z 456.484,A -85,B 0,C 180,E1 -6864.113,E2 -6864.113} C_VEL
LIN {X 0,Y 481.747,Z 456.478,A -85,B 0,C 180,E1 -6867.139,E2 -6867.139} C_VEL
LIN {X 0,Y 481.679,Z 456.488,A -85,B 0,C 180,E1 -6869.741,E2 -6869.741} C_VEL
LIN {X 0,Y 481.673,Z 456.485,A -85,B 0,C 180,E1 -6872.674,E2 -6872.674} C_VEL
LIN {X 0,Y 481.643,Z 456.491,A -85,B 0,C 180,E1 -6875.709,E2 -6875.709} C_VEL
LIN {X 0,Y 481.671,Z 456.486,A -85,B 0,C 180,E1 -6878.859,E2 -6878.859} C_VEL
LIN {X 0,Y 481.675,Z 456.487,A -85,B 0,C 180,E1 -6882.158,E2 -6882.158} C_VEL
LIN {X 0,Y 481.656,Z 456.49,A -85,B 0,C 180,E1 -6884.458,E2 -6884.458} C_VEL
LIN {X 0,Y 481.648,Z 456.491,A -85,B 0,C 180,E1 -6887.839,E2 -6887.839} C_VEL
LIN {X 0,Y 481.717,Z 456.634,A -85,B 0,C 180,E1 -6889.999,E2 -6889.999} C_VEL
LIN {X 0,Y 483.013,Z 463.994,A -85,B 0,C 180,E1 -6893.156,E2 -6893.156} C_VEL
LIN {X 0,Y 483.334,Z 467.32,A -85,B 0,C 180,E1 -6894.516,E2 -6894.516} C_VEL
LIN {X 0,Y 482.912,Z 475.266,A -85,B 0,C 180,E1 -6897.575,E2 -6897.575} C_VEL
LIN {X 0,Y 482.527,Z 482.625,A -85,B 0,C 180,E1 -6900.317,E2 -6900.317} C_VEL
LIN {X 0,Y 482.194,Z 490.414,A -85,B 0,C 180,E1 -6903.139,E2 -6903.139} C_VEL
LIN {X 0,Y 481.856,Z 499.554,A -85,B 0,C 180,E1 -6906.354,E2 -6906.354} C_VEL
LIN {X 0,Y 481.539,Z 508.718,A -85,B 0,C 180,E1 -6909.496,E2 -6909.496} C_VEL
LIN {X 0,Y 481.35,Z 516.607,A -85,B 0,C 180,E1 -6912.145,E2 -6912.145} C_VEL
LIN {X 0,Y 481.206,Z 525.524,A -85,B 0,C 180,E1 -6915.084,E2 -6915.084} C_VEL
LIN {X 0,Y 483.109,Z 538.991,A -85,B 0,C 180,E1 -6915.494,E2 -6915.494} C_VEL
LIN {X 0,Y 483.727,Z 544.269,A -85,B 0,C 180,E1 -6915.701,E2 -6915.701} C_VEL
LIN {X 0,Y 483.382,Z 556.102,A -85,B 0,C 180,E1 -6916.227,E2 -6916.227} C_VEL
LIN {X 0,Y 483.004,Z 567.438,A -85,B 0,C 180,E1 -6916.891,E2 -6916.891} C_VEL
LIN {X 0,Y 482.487,Z 579.718,A -85,B 0,C 180,E1 -6917.809,E2 -6917.809} C_VEL
LIN {X 0,Y 482.083,Z 589.795,A -85,B 0,C 180,E1 -6918.756,E2 -6918.756} C_VEL
LIN {X 0,Y 481.628,Z 599.76,A -85,B 0,C 180,E1 -6919.915,E2 -6919.915} C_VEL
LIN {X 0,Y 481.333,Z 608.555,A -85,B 0,C 180,E1 -6921.181,E2 -6921.181} C_VEL
LIN {X 0,Y 481.107,Z 615.572,A -85,B 0,C 180,E1 -6922.446,E2 -6922.446} C_VEL
LIN {X 0,Y 480.938,Z 621.583,A -85,B 0,C 180,E1 -6923.809,E2 -6923.809} C_VEL
LIN {X 0,Y 480.905,Z 625.602,A -85,B 0,C 180,E1 -6924.97,E2 -6924.97} C_VEL
LIN {X 0,Y 480.857,Z 627.928,A -85,B 0,C 180,E1 -6925.809,E2 -6925.809} C_VEL
LIN {X 0,Y 480.894,Z 629.822,A -85,B 0,C 180,E1 -6926.649,E2 -6926.649} C_VEL
LIN {X 0,Y 480.869,Z 631.238,A -85,B 0,C 180,E1 -6927.487,E2 -6927.487} C_VEL
LIN {X 0,Y 480.824,Z 632.239,A -85,B 0,C 180,E1 -6928.325,E2 -6928.325} C_VEL
LIN {X 0,Y 480.742,Z 633.044,A -85,B 0,C 180,E1 -6930,E2 -6930} C_VEL
LIN {X 0,Y 480.76,Z 632.811,A -85,B 0,C 180,E1 -6930.838,E2 -6930.838} C_VEL
LIN {X 0,Y 480.825,Z 632.176,A -85,B 0,C 180,E1 -6931.675,E2 -6931.675} C_VEL
LIN {X 0,Y 480.881,Z 631.138,A -85,B 0,C 180,E1 -6932.513,E2 -6932.513} C_VEL
LIN {X 0,Y 480.894,Z 629.685,A -85,B 0,C 180,E1 -6933.351,E2 -6933.351} C_VEL
LIN {X 0,Y 480.853,Z 626.642,A -85,B 0,C 180,E1 -6934.611,E2 -6934.611} C_VEL
LIN {X 0,Y 480.953,Z 622.537,A -85,B 0,C 180,E1 -6935.871,E2 -6935.871} C_VEL
LIN {X 0,Y 481.108,Z 616.223,A -85,B 0,C 180,E1 -6937.344,E2 -6937.344} C_VEL
LIN {X 0,Y 481.303,Z 609.328,A -85,B 0,C 180,E1 -6938.608,E2 -6938.608} C_VEL
LIN {X 0,Y 481.537,Z 600.774,A -85,B 0,C 180,E1 -6939.875,E2 -6939.875} C_VEL
LIN {X 0,Y 481.902,Z 591.98,A -85,B 0,C 180,E1 -6940.929,E2 -6940.929} C_VEL
LIN {X 0,Y 482.321,Z 581.319,A -85,B 0,C 180,E1 -6941.972,E2 -6941.972} C_VEL
LIN {X 0,Y 482.723,Z 570.801,A -85,B 0,C 180,E1 -6942.807,E2 -6942.807} C_VEL
LIN {X 0,Y 483.148,Z 558.748,A -85,B 0,C 180,E1 -6943.566,E2 -6943.566} C_VEL
LIN {X 0,Y 483.574,Z 545.484,A -85,B 0,C 180,E1 -6944.197,E2 -6944.197} C_VEL
LIN {X 0,Y 483.22,Z 540.186,A -85,B 0,C 180,E1 -6944.409,E2 -6944.409} C_VEL
LIN {X 0,Y 481.464,Z 526.603,A -85,B 0,C 180,E1 -6944.855,E2 -6944.855} C_VEL
LIN {X 0,Y 481.177,Z 524.249,A -85,B 0,C 180,E1 -6944.918,E2 -6944.918} C_VEL
LIN {X 0,Y 481.251,Z 515.065,A -85,B 0,C 180,E1 -6947.859,E2 -6947.859} C_VEL
LIN {X 0,Y 481.488,Z 505.759,A -85,B 0,C 180,E1 -6950.905,E2 -6950.905} C_VEL
LIN {X 0,Y 481.688,Z 496.306,A -85,B 0,C 180,E1 -6954.113,E2 -6954.113} C_VEL
LIN {X 0,Y 482.022,Z 487.666,A -85,B 0,C 180,E1 -6957.202,E2 -6957.202} C_VEL
LIN {X 0,Y 482.373,Z 479.924,A -85,B 0,C 180,E1 -6960.176,E2 -6960.176} C_VEL
LIN {X 0,Y 482.874,Z 473.051,A -85,B 0,C 180,E1 -6963.079,E2 -6963.079} C_VEL
LIN {X 0,Y 483.32,Z 467.859,A -85,B 0,C 180,E1 -6965.567,E2 -6965.567} C_VEL
LIN {X 0,Y 483.222,Z 465.5,A -85,B 0,C 180,E1 -6966.877,E2 -6966.877} C_VEL
LIN {X 0,Y 482.593,Z 461.645,A -85,B 0,C 180,E1 -6969.481,E2 -6969.481} C_VEL
LIN {X 0,Y 482.074,Z 458.808,A -85,B 0,C 180,E1 -6972.115,E2 -6972.115} C_VEL
LIN {X 0,Y 481.787,Z 457.245,A -85,B 0,C 180,E1 -6974.443,E2 -6974.443} C_VEL
LIN {X 0,Y 481.673,Z 456.489,A -85,B 0,C 180,E1 -6976.848,E2 -6976.848} C_VEL
LIN {X 0,Y 481.68,Z 456.602,A -85,B 0,C 180,E1 -6980.06,E2 -6980.06} C_VEL
LIN {X 0,Y 481.774,Z 457.262,A -85,B 0,C 180,E1 -6982.216,E2 -6982.216} C_VEL
LIN {X 0,Y 481.852,Z 458.489,A -85,B 0,C 180,E1 -6984.764,E2 -6984.764} C_VEL
LIN {X 0,Y 481.721,Z 460.097,A -85,B 0,C 180,E1 -6987.33,E2 -6987.33} C_VEL
LIN {X 0,Y 481.564,Z 462.204,A -85,B 0,C 180,E1 -6990.251,E2 -6990.251} C_VEL
LIN {X 0,Y 481.44,Z 464.478,A -85,B 0,C 180,E1 -6993.094,E2 -6993.094} C_VEL
LIN {X 0,Y 481.29,Z 466.84,A -85,B 0,C 180,E1 -6995.866,E2 -6995.866} C_VEL
LIN {X 0,Y 481.221,Z 470.102,A -85,B 0,C 180,E1 -6999.482,E2 -6999.482} C_VEL
LIN {X 0,Y 481.133,Z 472.621,A -85,B 0,C 180,E1 -7002.137,E2 -7002.137} C_VEL
LIN {X 0,Y 481.111,Z 475.839,A -85,B 0,C 180,E1 -7005.23,E2 -7005.23} C_VEL
LIN {X 0,Y 483.747,Z 487.707,A -85,B 0,C 180,E1 -7005.684,E2 -7005.684} C_VEL
LIN {X 0,Y 483.729,Z 499.221,A -85,B 0,C 180,E1 -7006.183,E2 -7006.183} C_VEL
LIN {X 0,Y 483.341,Z 510.544,A -85,B 0,C 180,E1 -7006.816,E2 -7006.816} C_VEL
LIN {X 0,Y 482.992,Z 521.613,A -85,B 0,C 180,E1 -7007.606,E2 -7007.606} C_VEL
LIN {X 0,Y 482.508,Z 532.207,A -85,B 0,C 180,E1 -7008.553,E2 -7008.553} C_VEL
LIN {X 0,Y 482.148,Z 540.883,A -85,B 0,C 180,E1 -7009.502,E2 -7009.502} C_VEL
LIN {X 0,Y 481.838,Z 548.863,A -85,B 0,C 180,E1 -7010.556,E2 -7010.556} C_VEL
LIN {X 0,Y 481.496,Z 556.698,A -85,B 0,C 180,E1 -7011.818,E2 -7011.818} C_VEL
LIN {X 0,Y 481.284,Z 561.989,A -85,B 0,C 180,E1 -7012.87,E2 -7012.87} C_VEL
LIN {X 0,Y 481.145,Z 567.147,A -85,B 0,C 180,E1 -7014.132,E2 -7014.132} C_VEL
LIN {X 0,Y 481.009,Z 571.138,A -85,B 0,C 180,E1 -7015.391,E2 -7015.391} C_VEL
LIN {X 0,Y 480.922,Z 574.074,A -85,B 0,C 180,E1 -7016.649,E2 -7016.649} C_VEL
LIN {X 0,Y 480.928,Z 575.488,A -85,B 0,C 180,E1 -7017.488,E2 -7017.488} C_VEL
LIN {X 0,Y 480.76,Z 577.088,A -85,B 0,C 180,E1 -7019.163,E2 -7019.163} C_VEL
LIN {X 0,Y 480.744,Z 577.307,A -85,B 0,C 180,E1 -7020,E2 -7020} C_VEL
LIN {X 0,Y 480.76,Z 577.099,A -85,B 0,C 180,E1 -7020.838,E2 -7020.838} C_VEL
LIN {X 0,Y 480.926,Z 575.483,A -85,B 0,C 180,E1 -7022.513,E2 -7022.513} C_VEL
LIN {X 0,Y 480.913,Z 574.091,A -85,B 0,C 180,E1 -7023.351,E2 -7023.351} C_VEL
LIN {X 0,Y 481.003,Z 571.16,A -85,B 0,C 180,E1 -7024.61,E2 -7024.61} C_VEL
LIN {X 0,Y 481.182,Z 566.177,A -85,B 0,C 180,E1 -7026.14,E2 -7026.14} C_VEL
LIN {X 0,Y 481.302,Z 560.075,A -85,B 0,C 180,E1 -7027.552,E2 -7027.552} C_VEL
LIN {X 0,Y 481.599,Z 553.167,A -85,B 0,C 180,E1 -7028.814,E2 -7028.814} C_VEL
LIN {X 0,Y 481.939,Z 544.51,A -85,B 0,C 180,E1 -7030.079,E2 -7030.079} C_VEL
LIN {X 0,Y 482.304,Z 535.641,A -85,B 0,C 180,E1 -7031.133,E2 -7031.133} C_VEL
LIN {X 0,Y 482.769,Z 525.91,A -85,B 0,C 180,E1 -7032.08,E2 -7032.08} C_VEL
LIN {X 0,Y 483.06,Z 515.7,A -85,B 0,C 180,E1 -7032.895,E2 -7032.895} C_VEL
LIN {X 0,Y 483.493,Z 503.394,A -85,B 0,C 180,E1 -7033.663,E2 -7033.663} C_VEL
LIN {X 0,Y 483.858,Z 491.187,A -85,B 0,C 180,E1 -7034.242,E2 -7034.242} C_VEL
LIN {X 0,Y 483.271,Z 484.851,A -85,B 0,C 180,E1 -7034.502,E2 -7034.502} C_VEL
LIN {X 0,Y 480.957,Z 474.164,A -85,B 0,C 180,E1 -7034.898,E2 -7034.898} C_VEL
LIN {X 0,Y 480.962,Z 470.439,A -85,B 0,C 180,E1 -7038.23,E2 -7038.23} C_VEL
LIN {X 0,Y 480.953,Z 466.935,A -85,B 0,C 180,E1 -7041.427,E2 -7041.427} C_VEL
LIN {X 0,Y 480.988,Z 463.983,A -85,B 0,C 180,E1 -7044.15,E2 -7044.15} C_VEL
LIN {X 0,Y 481.089,Z 460.952,A -85,B 0,C 180,E1 -7046.985,E2 -7046.985} C_VEL
LIN {X 0,Y 481.117,Z 457.981,A -85,B 0,C 180,E1 -7049.78,E2 -7049.78} C_VEL
LIN {X 0,Y 481.127,Z 456.96,A -85,B 0,C 180,E1 -7050.748,E2 -7050.748} C_VEL
LIN {X 0,Y 481.22,Z 456.546,A -85,B 0,C 180,E1 -7052.106,E2 -7052.106} C_VEL
LIN {X 0,Y 481.566,Z 456.5,A -85,B 0,C 180,E1 -7055.187,E2 -7055.187} C_VEL
LIN {X 0,Y 481.654,Z 456.488,A -85,B 0,C 180,E1 -7058.007,E2 -7058.007} C_VEL
LIN {X 0,Y 481.662,Z 456.488,A -85,B 0,C 180,E1 -7061.042,E2 -7061.042} C_VEL
LIN {X 0,Y 481.66,Z 456.491,A -85,B 0,C 180,E1 -7064.458,E2 -7064.458} C_VEL
LIN {X 0,Y 481.652,Z 456.491,A -85,B 0,C 180,E1 -7067.839,E2 -7067.839} C_VEL
LIN {X 0,Y 481.686,Z 456.487,A -85,B 0,C 180,E1 -7070.651,E2 -7070.651} C_VEL
LIN {X 0,Y 481.633,Z 456.489,A -85,B 0,C 180,E1 -7073.376,E2 -7073.376} C_VEL
LIN {X 0,Y 481.715,Z 456.481,A -85,B 0,C 180,E1 -7076.33,E2 -7076.33} C_VEL
LIN {X 0,Y 481.655,Z 456.487,A -85,B 0,C 180,E1 -7079.418,E2 -7079.418} C_VEL
LIN {X 0,Y 481.704,Z 456.483,A -85,B 0,C 180,E1 -7082.168,E2 -7082.168} C_VEL
LIN {X 0,Y 481.706,Z 456.481,A -85,B 0,C 180,E1 -7083.987,E2 -7083.987} C_VEL
LIN {X 0,Y 481.047,Z 456.566,A -85,B 0,C 180,E1 -7084.685,E2 -7084.685} C_VEL
LIN {X 0,Y 478.175,Z 456.923,A -85,B 0,C 180,E1 -7085.817,E2 -7085.817} C_VEL
LIN {X 0,Y 475.733,Z 457.225,A -85,B 0,C 180,E1 -7086.731,E2 -7086.731} C_VEL
LIN {X 0,Y 474.678,Z 457.355,A -85,B 0,C 180,E1 -7087.437,E2 -7087.437} C_VEL
LIN {X 0,Y 474.588,Z 457.366,A -85,B 0,C 180,E1 -7087.676,E2 -7087.676} C_VEL
LIN {X 0,Y 474.661,Z 457.36,A -85,B 0,C 180,E1 -7090.09,E2 -7090.09} C_VEL
LIN {X 0,Y 474.653,Z 457.361,A -85,B 0,C 180,E1 -7092.774,E2 -7092.774} C_VEL
LIN {X 0,Y 474.655,Z 457.359,A -85,B 0,C 180,E1 -7095.421,E2 -7095.421} C_VEL
LIN {X 0,Y 474.711,Z 457.353,A -85,B 0,C 180,E1 -7098.038,E2 -7098.038} C_VEL
LIN {X 0,Y 474.717,Z 457.351,A -85,B 0,C 180,E1 -7101.486,E2 -7101.486} C_VEL
LIN {X 0,Y 474.784,Z 457.345,A -85,B 0,C 180,E1 -7104.052,E2 -7104.052} C_VEL
LIN {X 0,Y 474.899,Z 457.329,A -85,B 0,C 180,E1 -7107.455,E2 -7107.455} C_VEL
LIN {X 0,Y 474.918,Z 457.33,A -85,B 0,C 180,E1 -7110,E2 -7110} C_VEL
LIN {X 0,Y 474.899,Z 457.331,A -85,B 0,C 180,E1 -7112.544,E2 -7112.544} C_VEL
LIN {X 0,Y 474.764,Z 457.349,A -85,B 0,C 180,E1 -7115.948,E2 -7115.948} C_VEL
LIN {X 0,Y 474.734,Z 457.35,A -85,B 0,C 180,E1 -7118.513,E2 -7118.513} C_VEL
LIN {X 0,Y 474.71,Z 457.355,A -85,B 0,C 180,E1 -7121.962,E2 -7121.962} C_VEL
LIN {X 0,Y 474.705,Z 457.356,A -85,B 0,C 180,E1 -7125.455,E2 -7125.455} C_VEL
LIN {X 0,Y 474.67,Z 457.358,A -85,B 0,C 180,E1 -7129.01,E2 -7129.01} C_VEL
LIN {X 0,Y 474.594,Z 457.371,A -85,B 0,C 180,E1 -7131.728,E2 -7131.728} C_VEL
LIN {X 0,Y 474.662,Z 457.361,A -85,B 0,C 180,E1 -7134.493,E2 -7134.493} C_VEL
LIN {X 0,Y 474.685,Z 457.355,A -85,B 0,C 180,E1 -7137.334,E2 -7137.334} C_VEL
LIN {X 0,Y 474.609,Z 457.365,A -85,B 0,C 180,E1 -7140.23,E2 -7140.23} C_VEL
LIN {X 0,Y 474.647,Z 457.361,A -85,B 0,C 180,E1 -7143.22,E2 -7143.22} C_VEL
LIN {X 0,Y 474.596,Z 457.366,A -85,B 0,C 180,E1 -7146.323,E2 -7146.323} C_VEL
LIN {X 0,Y 474.631,Z 457.363,A -85,B 0,C 180,E1 -7149.647,E2 -7149.647} C_VEL
LIN {X 0,Y 474.618,Z 457.363,A -85,B 0,C 180,E1 -7152.934,E2 -7152.934} C_VEL
LIN {X 0,Y 474.618,Z 457.365,A -85,B 0,C 180,E1 -7155.895,E2 -7155.895} C_VEL
LIN {X 0,Y 474.635,Z 457.361,A -85,B 0,C 180,E1 -7159.04,E2 -7159.04} C_VEL
LIN {X 0,Y 474.613,Z 457.366,A -85,B 0,C 180,E1 -7161.704,E2 -7161.704} C_VEL
LIN {X 0,Y 474.632,Z 457.363,A -85,B 0,C 180,E1 -7164.726,E2 -7164.726} C_VEL
LIN {X 0,Y 474.638,Z 457.363,A -85,B 0,C 180,E1 -7167.787,E2 -7167.787} C_VEL
LIN {X 0,Y 474.626,Z 457.365,A -85,B 0,C 180,E1 -7170.884,E2 -7170.884} C_VEL
LIN {X 0,Y 474.663,Z 457.362,A -85,B 0,C 180,E1 -7173.628,E2 -7173.628} C_VEL
LIN {X 0,Y 474.637,Z 457.363,A -85,B 0,C 180,E1 -7176.641,E2 -7176.641} C_VEL
LIN {X 0,Y 474.658,Z 457.361,A -85,B 0,C 180,E1 -7180.089,E2 -7180.089} C_VEL
LIN {X 0,Y 474.652,Z 457.36,A -85,B 0,C 180,E1 -7182.774,E2 -7182.774} C_VEL
LIN {X 0,Y 474.65,Z 457.361,A -85,B 0,C 180,E1 -7185.421,E2 -7185.421} C_VEL
LIN {X 0,Y 474.706,Z 457.353,A -85,B 0,C 180,E1 -7188.037,E2 -7188.037} C_VEL
LIN {X 0,Y 474.73,Z 457.351,A -85,B 0,C 180,E1 -7191.486,E2 -7191.486} C_VEL
LIN {X 0,Y 474.78,Z 457.346,A -85,B 0,C 180,E1 -7194.052,E2 -7194.052} C_VEL
LIN {X 0,Y 474.895,Z 457.332,A -85,B 0,C 180,E1 -7197.455,E2 -7197.455} C_VEL
LIN {X 0,Y 474.913,Z 457.33,A -85,B 0,C 180,E1 -7200,E2 -7200} C_VEL
LIN {X 0,Y 474.895,Z 457.328,A -85,B 0,C 180,E1 -7202.544,E2 -7202.544} C_VEL
LIN {X 0,Y 474.78,Z 457.345,A -85,B 0,C 180,E1 -7205.947,E2 -7205.947} C_VEL
LIN {X 0,Y 474.729,Z 457.351,A -85,B 0,C 180,E1 -7208.513,E2 -7208.513} C_VEL
LIN {X 0,Y 474.705,Z 457.353,A -85,B 0,C 180,E1 -7211.962,E2 -7211.962} C_VEL
LIN {X 0,Y 474.701,Z 457.355,A -85,B 0,C 180,E1 -7215.456,E2 -7215.456} C_VEL
LIN {X 0,Y 474.666,Z 457.361,A -85,B 0,C 180,E1 -7219.01,E2 -7219.01} C_VEL
LIN {X 0,Y 474.59,Z 457.37,A -85,B 0,C 180,E1 -7221.729,E2 -7221.729} C_VEL
LIN {X 0,Y 474.66,Z 457.357,A -85,B 0,C 180,E1 -7224.493,E2 -7224.493} C_VEL
LIN {X 0,Y 474.7,Z 457.355,A -85,B 0,C 180,E1 -7227.339,E2 -7227.339} C_VEL
LIN {X 0,Y 474.604,Z 457.365,A -85,B 0,C 180,E1 -7230.81,E2 -7230.81} C_VEL
LIN {X 0,Y 474.639,Z 457.362,A -85,B 0,C 180,E1 -7233.984,E2 -7233.984} C_VEL
LIN {X 0,Y 474.575,Z 457.37,A -85,B 0,C 180,E1 -7236.9,E2 -7236.9} C_VEL
LIN {X 0,Y 474.628,Z 457.363,A -85,B 0,C 180,E1 -7239.648,E2 -7239.648} C_VEL
LIN {X 0,Y 474.653,Z 457.361,A -85,B 0,C 180,E1 -7242.93,E2 -7242.93} C_VEL
LIN {X 0,Y 474.606,Z 457.371,A -85,B 0,C 180,E1 -7245.895,E2 -7245.895} C_VEL
LIN {X 0,Y 474.628,Z 457.367,A -85,B 0,C 180,E1 -7249.041,E2 -7249.041} C_VEL
LIN {X 0,Y 474.669,Z 457.509,A -85,B 0,C 180,E1 -7249.738,E2 -7249.738} C_VEL
LIN {X 0,Y 475.94,Z 464.704,A -85,B 0,C 180,E1 -7252.882,E2 -7252.882} C_VEL
LIN {X 0,Y 476.344,Z 467.954,A -85,B 0,C 180,E1 -7254.24,E2 -7254.24} C_VEL
LIN {X 0,Y 475.931,Z 475.808,A -85,B 0,C 180,E1 -7257.321,E2 -7257.321} C_VEL
LIN {X 0,Y 475.508,Z 483.715,A -85,B 0,C 180,E1 -7260.321,E2 -7260.321} C_VEL
LIN {X 0,Y 475.139,Z 491.509,A -85,B 0,C 180,E1 -7263.183,E2 -7263.183} C_VEL
LIN {X 0,Y 474.785,Z 500.617,A -85,B 0,C 180,E1 -7266.443,E2 -7266.443} C_VEL
LIN {X 0,Y 474.473,Z 509.767,A -85,B 0,C 180,E1 -7269.63,E2 -7269.63} C_VEL
LIN {X 0,Y 474.275,Z 517.621,A -85,B 0,C 180,E1 -7272.316,E2 -7272.316} C_VEL
LIN {X 0,Y 474.166,Z 525.159,A -85,B 0,C 180,E1 -7274.857,E2 -7274.857} C_VEL
LIN {X 0,Y 476.158,Z 539.63,A -85,B 0,C 180,E1 -7275.318,E2 -7275.318} C_VEL
LIN {X 0,Y 476.792,Z 545.091,A -85,B 0,C 180,E1 -7275.543,E2 -7275.543} C_VEL
LIN {X 0,Y 476.379,Z 557.526,A -85,B 0,C 180,E1 -7276.129,E2 -7276.129} C_VEL
LIN {X 0,Y 475.926,Z 569.574,A -85,B 0,C 180,E1 -7276.878,E2 -7276.878} C_VEL
LIN {X 0,Y 475.43,Z 580.796,A -85,B 0,C 180,E1 -7277.765,E2 -7277.765} C_VEL
LIN {X 0,Y 475.031,Z 590.294,A -85,B 0,C 180,E1 -7278.695,E2 -7278.695} C_VEL
LIN {X 0,Y 474.593,Z 599.292,A -85,B 0,C 180,E1 -7279.764,E2 -7279.764} C_VEL
LIN {X 0,Y 474.271,Z 608.104,A -85,B 0,C 180,E1 -7281.049,E2 -7281.049} C_VEL
LIN {X 0,Y 474.038,Z 615.138,A -85,B 0,C 180,E1 -7282.332,E2 -7282.332} C_VEL
LIN {X 0,Y 473.879,Z 620.512,A -85,B 0,C 180,E1 -7283.547,E2 -7283.547} C_VEL
LIN {X 0,Y 473.839,Z 625.188,A -85,B 0,C 180,E1 -7284.895,E2 -7284.895} C_VEL
LIN {X 0,Y 473.76,Z 627.516,A -85,B 0,C 180,E1 -7285.746,E2 -7285.746} C_VEL
LIN {X 0,Y 473.82,Z 629.414,A -85,B 0,C 180,E1 -7286.599,E2 -7286.599} C_VEL
LIN {X 0,Y 473.783,Z 630.833,A -85,B 0,C 180,E1 -7287.45,E2 -7287.45} C_VEL
LIN {X 0,Y 473.758,Z 631.834,A -85,B 0,C 180,E1 -7288.3,E2 -7288.3} C_VEL
LIN {X 0,Y 473.688,Z 632.434,A -85,B 0,C 180,E1 -7289.15,E2 -7289.15} C_VEL
LIN {X 0,Y 473.669,Z 632.636,A -85,B 0,C 180,E1 -7290,E2 -7290} C_VEL
LIN {X 0,Y 473.688,Z 632.399,A -85,B 0,C 180,E1 -7290.85,E2 -7290.85} C_VEL
LIN {X 0,Y 473.758,Z 631.755,A -85,B 0,C 180,E1 -7291.7,E2 -7291.7} C_VEL
LIN {X 0,Y 473.793,Z 630.71,A -85,B 0,C 180,E1 -7292.551,E2 -7292.551} C_VEL
LIN {X 0,Y 473.821,Z 629.249,A -85,B 0,C 180,E1 -7293.402,E2 -7293.402} C_VEL
LIN {X 0,Y 473.775,Z 626.188,A -85,B 0,C 180,E1 -7294.68,E2 -7294.68} C_VEL
LIN {X 0,Y 473.859,Z 622.06,A -85,B 0,C 180,E1 -7295.959,E2 -7295.959} C_VEL
LIN {X 0,Y 474.017,Z 615.709,A -85,B 0,C 180,E1 -7297.454,E2 -7297.454} C_VEL
LIN {X 0,Y 474.213,Z 608.785,A -85,B 0,C 180,E1 -7298.738,E2 -7298.738} C_VEL
LIN {X 0,Y 474.495,Z 600.203,A -85,B 0,C 180,E1 -7300.023,E2 -7300.023} C_VEL
LIN {X 0,Y 474.897,Z 591.38,A -85,B 0,C 180,E1 -7301.092,E2 -7301.092} C_VEL
LIN {X 0,Y 475.329,Z 580.967,A -85,B 0,C 180,E1 -7302.126,E2 -7302.126} C_VEL
LIN {X 0,Y 475.79,Z 569.873,A -85,B 0,C 180,E1 -7303.018,E2 -7303.018} C_VEL
LIN {X 0,Y 476.213,Z 558.093,A -85,B 0,C 180,E1 -7303.767,E2 -7303.767} C_VEL
LIN {X 0,Y 476.671,Z 544.882,A -85,B 0,C 180,E1 -7304.407,E2 -7304.407} C_VEL
LIN {X 0,Y 475.105,Z 531.592,A -85,B 0,C 180,E1 -7304.921,E2 -7304.921} C_VEL
LIN {X 0,Y 474.095,Z 523.676,A -85,B 0,C 180,E1 -7305.173,E2 -7305.173} C_VEL
LIN {X 0,Y 474.241,Z 513.586,A -85,B 0,C 180,E1 -7308.478,E2 -7308.478} C_VEL
LIN {X 0,Y 474.466,Z 503.913,A -85,B 0,C 180,E1 -7311.735,E2 -7311.735} C_VEL
LIN {X 0,Y 474.736,Z 494.736,A -85,B 0,C 180,E1 -7314.956,E2 -7314.956} C_VEL
LIN {X 0,Y 475.041,Z 487.111,A -85,B 0,C 180,E1 -7317.786,E2 -7317.786} C_VEL
LIN {X 0,Y 475.545,Z 478.739,A -85,B 0,C 180,E1 -7321.149,E2 -7321.149} C_VEL
LIN {X 0,Y 476.132,Z 471.877,A -85,B 0,C 180,E1 -7324.249,E2 -7324.249} C_VEL
LIN {X 0,Y 476.32,Z 468.198,A -85,B 0,C 180,E1 -7326.171,E2 -7326.171} C_VEL
LIN {X 0,Y 475.913,Z 464.511,A -85,B 0,C 180,E1 -7328.494,E2 -7328.494} C_VEL
LIN {X 0,Y 475.366,Z 461.397,A -85,B 0,C 180,E1 -7331.062,E2 -7331.062} C_VEL
LIN {X 0,Y 474.941,Z 459.348,A -85,B 0,C 180,E1 -7333.524,E2 -7333.524} C_VEL
LIN {X 0,Y 474.745,Z 458.223,A -85,B 0,C 180,E1 -7335.911,E2 -7335.911} C_VEL
LIN {X 0,Y 474.712,Z 457.857,A -85,B 0,C 180,E1 -7338.224,E2 -7338.224} C_VEL
LIN {X 0,Y 474.719,Z 458.081,A -85,B 0,C 180,E1 -7340.462,E2 -7340.462} C_VEL
LIN {X 0,Y 474.805,Z 458.912,A -85,B 0,C 180,E1 -7343.064,E2 -7343.064} C_VEL
LIN {X 0,Y 474.789,Z 460.268,A -85,B 0,C 180,E1 -7345.772,E2 -7345.772} C_VEL
LIN {X 0,Y 474.629,Z 462.195,A -85,B 0,C 180,E1 -7348.785,E2 -7348.785} C_VEL
LIN {X 0,Y 474.456,Z 464.361,A -85,B 0,C 180,E1 -7351.705,E2 -7351.705} C_VEL
LIN {X 0,Y 474.315,Z 466.748,A -85,B 0,C 180,E1 -7354.669,E2 -7354.669} C_VEL
LIN {X 0,Y 474.177,Z 469.041,A -85,B 0,C 180,E1 -7357.334,E2 -7357.334} C_VEL
LIN {X 0,Y 474.091,Z 471.502,A -85,B 0,C 180,E1 -7360.065,E2 -7360.065} C_VEL
LIN {X 0,Y 474.043,Z 474.028,A -85,B 0,C 180,E1 -7362.752,E2 -7362.752} C_VEL
LIN {X 0,Y 474.039,Z 476.2,A -85,B 0,C 180,E1 -7364.985,E2 -7364.985} C_VEL
LIN {X 0,Y 476.869,Z 488.579,A -85,B 0,C 180,E1 -7365.49,E2 -7365.49} C_VEL
LIN {X 0,Y 476.863,Z 499.583,A -85,B 0,C 180,E1 -7365.98,E2 -7365.98} C_VEL
LIN {X 0,Y 476.456,Z 511.173,A -85,B 0,C 180,E1 -7366.639,E2 -7366.639} C_VEL
LIN {X 0,Y 476.075,Z 521.99,A -85,B 0,C 180,E1 -7367.424,E2 -7367.424} C_VEL
LIN {X 0,Y 475.573,Z 532.592,A -85,B 0,C 180,E1 -7368.384,E2 -7368.384} C_VEL
LIN {X 0,Y 475.183,Z 541.279,A -85,B 0,C 180,E1 -7369.346,E2 -7369.346} C_VEL
LIN {X 0,Y 474.85,Z 549.269,A -85,B 0,C 180,E1 -7370.415,E2 -7370.415} C_VEL
LIN {X 0,Y 474.475,Z 557.108,A -85,B 0,C 180,E1 -7371.697,E2 -7371.697} C_VEL
LIN {X 0,Y 474.248,Z 562.398,A -85,B 0,C 180,E1 -7372.764,E2 -7372.764} C_VEL
LIN {X 0,Y 474.102,Z 567.557,A -85,B 0,C 180,E1 -7374.044,E2 -7374.044} C_VEL
LIN {X 0,Y 473.947,Z 571.551,A -85,B 0,C 180,E1 -7375.322,E2 -7375.322} C_VEL
LIN {X 0,Y 473.856,Z 574.488,A -85,B 0,C 180,E1 -7376.599,E2 -7376.599} C_VEL
LIN {X 0,Y 473.868,Z 575.904,A -85,B 0,C 180,E1 -7377.45,E2 -7377.45} C_VEL
LIN {X 0,Y 473.689,Z 577.502,A -85,B 0,C 180,E1 -7379.15,E2 -7379.15} C_VEL
LIN {X 0,Y 473.671,Z 577.718,A -85,B 0,C 180,E1 -7380,E2 -7380} C_VEL
LIN {X 0,Y 473.689,Z 577.507,A -85,B 0,C 180,E1 -7380.85,E2 -7380.85} C_VEL
LIN {X 0,Y 473.866,Z 575.875,A -85,B 0,C 180,E1 -7382.55,E2 -7382.55} C_VEL
LIN {X 0,Y 473.848,Z 574.476,A -85,B 0,C 180,E1 -7383.401,E2 -7383.401} C_VEL
LIN {X 0,Y 473.939,Z 571.53,A -85,B 0,C 180,E1 -7384.678,E2 -7384.678} C_VEL
LIN {X 0,Y 474.091,Z 567.545,A -85,B 0,C 180,E1 -7385.957,E2 -7385.957} C_VEL
LIN {X 0,Y 474.257,Z 561.411,A -85,B 0,C 180,E1 -7387.451,E2 -7387.451} C_VEL
LIN {X 0,Y 474.511,Z 554.704,A -85,B 0,C 180,E1 -7388.732,E2 -7388.732} C_VEL
LIN {X 0,Y 474.867,Z 546.385,A -85,B 0,C 180,E1 -7390.015,E2 -7390.015} C_VEL
LIN {X 0,Y 475.198,Z 537.831,A -85,B 0,C 180,E1 -7391.085,E2 -7391.085} C_VEL
LIN {X 0,Y 475.783,Z 527.293,A -85,B 0,C 180,E1 -7392.152,E2 -7392.152} C_VEL
LIN {X 0,Y 476.125,Z 516.511,A -85,B 0,C 180,E1 -7393.038,E2 -7393.038} C_VEL
LIN {X 0,Y 476.534,Z 505.489,A -85,B 0,C 180,E1 -7393.758,E2 -7393.758} C_VEL
LIN {X 0,Y 476.947,Z 492.57,A -85,B 0,C 180,E1 -7394.399,E2 -7394.399} C_VEL
LIN {X 0,Y 476.548,Z 486.903,A -85,B 0,C 180,E1 -7394.638,E2 -7394.638} C_VEL
LIN {X 0,Y 473.91,Z 474.484,A -85,B 0,C 180,E1 -7395.115,E2 -7395.115} C_VEL
LIN {X 0,Y 473.905,Z 470.893,A -85,B 0,C 180,E1 -7398.355,E2 -7398.355} C_VEL
LIN {X 0,Y 473.882,Z 467.171,A -85,B 0,C 180,E1 -7401.763,E2 -7401.763} C_VEL
LIN {X 0,Y 473.925,Z 464.191,A -85,B 0,C 180,E1 -7404.534,E2 -7404.534} C_VEL
LIN {X 0,Y 474.021,Z 461.181,A -85,B 0,C 180,E1 -7407.363,E2 -7407.363} C_VEL
LIN {X 0,Y 474.061,Z 457.673,A -85,B 0,C 180,E1 -7410.699,E2 -7410.699} C_VEL
LIN {X 0,Y 474.312,Z 457.404,A -85,B 0,C 180,E1 -7413.247,E2 -7413.247} C_VEL
LIN {X 0,Y 474.545,Z 457.375,A -85,B 0,C 180,E1 -7415.457,E2 -7415.457} C_VEL
LIN {X 0,Y 474.614,Z 457.367,A -85,B 0,C 180,E1 -7418.458,E2 -7418.458} C_VEL
LIN {X 0,Y 474.633,Z 457.363,A -85,B 0,C 180,E1 -7420.959,E2 -7420.959} C_VEL
LIN {X 0,Y 474.611,Z 457.366,A -85,B 0,C 180,E1 -7424.105,E2 -7424.105} C_VEL
LIN {X 0,Y 474.619,Z 457.363,A -85,B 0,C 180,E1 -7427.066,E2 -7427.066} C_VEL
LIN {X 0,Y 474.65,Z 457.362,A -85,B 0,C 180,E1 -7430.454,E2 -7430.454} C_VEL
LIN {X 0,Y 474.594,Z 457.367,A -85,B 0,C 180,E1 -7433.677,E2 -7433.677} C_VEL
LIN {X 0,Y 474.648,Z 457.363,A -85,B 0,C 180,E1 -7436.78,E2 -7436.78} C_VEL
LIN {X 0,Y 474.609,Z 457.365,A -85,B 0,C 180,E1 -7439.77,E2 -7439.77} C_VEL
LIN {X 0,Y 474.703,Z 457.354,A -85,B 0,C 180,E1 -7442.68,E2 -7442.68} C_VEL
LIN {X 0,Y 474.663,Z 457.359,A -85,B 0,C 180,E1 -7445.507,E2 -7445.507} C_VEL
LIN {X 0,Y 474.588,Z 457.366,A -85,B 0,C 180,E1 -7447.676,E2 -7447.676} C_VEL
LIN {X 0,Y 473.916,Z 457.453,A -85,B 0,C 180,E1 -7448.384,E2 -7448.384} C_VEL
LIN {X 0,Y 471.08,Z 457.807,A -85,B 0,C 180,E1 -7449.535,E2 -7449.535} C_VEL
LIN {X 0,Y 468.701,Z 458.103,A -85,B 0,C 180,E1 -7450.464,E2 -7450.464} C_VEL
LIN {X 0,Y 467.7,Z 458.227,A -85,B 0,C 180,E1 -7451.18,E2 -7451.18} C_VEL
LIN {X 0,Y 467.628,Z 458.236,A -85,B 0,C 180,E1 -7451.423,E2 -7451.423} C_VEL
LIN {X 0,Y 467.645,Z 458.235,A -85,B 0,C 180,E1 -7454.305,E2 -7454.305} C_VEL
LIN {X 0,Y 467.662,Z 458.232,A -85,B 0,C 180,E1 -7457.855,E2 -7457.855} C_VEL
LIN {X 0,Y 467.675,Z 458.228,A -85,B 0,C 180,E1 -7461.357,E2 -7461.357} C_VEL
LIN {X 0,Y 467.748,Z 458.222,A -85,B 0,C 180,E1 -7463.962,E2 -7463.962} C_VEL
LIN {X 0,Y 467.865,Z 458.205,A -85,B 0,C 180,E1 -7467.417,E2 -7467.417} C_VEL
LIN {X 0,Y 467.888,Z 458.205,A -85,B 0,C 180,E1 -7470,E2 -7470} C_VEL
LIN {X 0,Y 467.864,Z 458.208,A -85,B 0,C 180,E1 -7472.583,E2 -7472.583} C_VEL
LIN {X 0,Y 467.726,Z 458.227,A -85,B 0,C 180,E1 -7476.037,E2 -7476.037} C_VEL
LIN {X 0,Y 467.687,Z 458.228,A -85,B 0,C 180,E1 -7478.642,E2 -7478.642} C_VEL
LIN {X 0,Y 467.662,Z 458.234,A -85,B 0,C 180,E1 -7482.145,E2 -7482.145} C_VEL
LIN {X 0,Y 467.645,Z 458.235,A -85,B 0,C 180,E1 -7485.695,E2 -7485.695} C_VEL
LIN {X 0,Y 467.622,Z 458.236,A -85,B 0,C 180,E1 -7488.764,E2 -7488.764} C_VEL
LIN {X 0,Y 467.585,Z 458.239,A -85,B 0,C 180,E1 -7491.268,E2 -7491.268} C_VEL
LIN {X 0,Y 467.577,Z 458.242,A -85,B 0,C 180,E1 -7493.943,E2 -7493.943} C_VEL
LIN {X 0,Y 467.621,Z 458.235,A -85,B 0,C 180,E1 -7496.8,E2 -7496.8} C_VEL
LIN {X 0,Y 467.558,Z 458.246,A -85,B 0,C 180,E1 -7499.738,E2 -7499.738} C_VEL
LIN {X 0,Y 467.587,Z 458.241,A -85,B 0,C 180,E1 -7502.758,E2 -7502.758} C_VEL
LIN {X 0,Y 467.56,Z 458.246,A -85,B 0,C 180,E1 -7505.889,E2 -7505.889} C_VEL
LIN {X 0,Y 467.585,Z 458.242,A -85,B 0,C 180,E1 -7509.144,E2 -7509.144} C_VEL
LIN {X 0,Y 467.589,Z 458.238,A -85,B 0,C 180,E1 -7512.567,E2 -7512.567} C_VEL
LIN {X 0,Y 467.574,Z 458.243,A -85,B 0,C 180,E1 -7515.053,E2 -7515.053} C_VEL
LIN {X 0,Y 467.591,Z 458.24,A -85,B 0,C 180,E1 -7517.44,E2 -7517.44} C_VEL
LIN {X 0,Y 467.562,Z 458.243,A -85,B 0,C 180,E1 -7520.853,E2 -7520.853} C_VEL
LIN {X 0,Y 467.565,Z 458.245,A -85,B 0,C 180,E1 -7524.26,E2 -7524.26} C_VEL
LIN {X 0,Y 467.584,Z 458.241,A -85,B 0,C 180,E1 -7527.32,E2 -7527.32} C_VEL
LIN {X 0,Y 467.572,Z 458.243,A -85,B 0,C 180,E1 -7530.667,E2 -7530.667} C_VEL
LIN {X 0,Y 467.618,Z 458.236,A -85,B 0,C 180,E1 -7533.199,E2 -7533.199} C_VEL
LIN {X 0,Y 467.594,Z 458.24,A -85,B 0,C 180,E1 -7536.468,E2 -7536.468} C_VEL
LIN {X 0,Y 467.626,Z 458.238,A -85,B 0,C 180,E1 -7539.777,E2 -7539.777} C_VEL
LIN {X 0,Y 467.611,Z 458.236,A -85,B 0,C 180,E1 -7542.507,E2 -7542.507} C_VEL
LIN {X 0,Y 467.608,Z 458.239,A -85,B 0,C 180,E1 -7545.196,E2 -7545.196} C_VEL
LIN {X 0,Y 467.657,Z 458.233,A -85,B 0,C 180,E1 -7547.854,E2 -7547.854} C_VEL
LIN {X 0,Y 467.683,Z 458.23,A -85,B 0,C 180,E1 -7551.357,E2 -7551.357} C_VEL
LIN {X 0,Y 467.745,Z 458.223,A -85,B 0,C 180,E1 -7553.962,E2 -7553.962} C_VEL
LIN {X 0,Y 467.86,Z 458.208,A -85,B 0,C 180,E1 -7557.417,E2 -7557.417} C_VEL
LIN {X 0,Y 467.884,Z 458.206,A -85,B 0,C 180,E1 -7560,E2 -7560} C_VEL
LIN {X 0,Y 467.86,Z 458.204,A -85,B 0,C 180,E1 -7562.583,E2 -7562.583} C_VEL
LIN {X 0,Y 467.745,Z 458.222,A -85,B 0,C 180,E1 -7566.037,E2 -7566.037} C_VEL
LIN {X 0,Y 467.682,Z 458.228,A -85,B 0,C 180,E1 -7568.643,E2 -7568.643} C_VEL
LIN {X 0,Y 467.657,Z 458.232,A -85,B 0,C 180,E1 -7572.145,E2 -7572.145} C_VEL
LIN {X 0,Y 467.64,Z 458.237,A -85,B 0,C 180,E1 -7575.695,E2 -7575.695} C_VEL
LIN {X 0,Y 467.618,Z 458.237,A -85,B 0,C 180,E1 -7578.765,E2 -7578.765} C_VEL
LIN {X 0,Y 467.581,Z 458.241,A -85,B 0,C 180,E1 -7581.268,E2 -7581.268} C_VEL
LIN {X 0,Y 467.574,Z 458.241,A -85,B 0,C 180,E1 -7583.943,E2 -7583.943} C_VEL
LIN {X 0,Y 467.617,Z 458.238,A -85,B 0,C 180,E1 -7586.8,E2 -7586.8} C_VEL
LIN {X 0,Y 467.554,Z 458.247,A -85,B 0,C 180,E1 -7589.738,E2 -7589.738} C_VEL
LIN {X 0,Y 467.584,Z 458.241,A -85,B 0,C 180,E1 -7592.758,E2 -7592.758} C_VEL
LIN {X 0,Y 467.557,Z 458.246,A -85,B 0,C 180,E1 -7595.889,E2 -7595.889} C_VEL
LIN {X 0,Y 467.583,Z 458.243,A -85,B 0,C 180,E1 -7599.145,E2 -7599.145} C_VEL
LIN {X 0,Y 467.62,Z 458.238,A -85,B 0,C 180,E1 -7602.571,E2 -7602.571} C_VEL
LIN {X 0,Y 467.552,Z 458.249,A -85,B 0,C 180,E1 -7606.179,E2 -7606.179} C_VEL
LIN {X 0,Y 467.585,Z 458.244,A -85,B 0,C 180,E1 -7609.312,E2 -7609.312} C_VEL
LIN {X 0,Y 468,Z 460.558,A -85,B 0,C 180,E1 -7610.463,E2 -7610.463} C_VEL
LIN {X 0,Y 469.102,Z 466.75,A -85,B 0,C 180,E1 -7613.182,E2 -7613.182} C_VEL
LIN {X 0,Y 469.334,Z 470.622,A -85,B 0,C 180,E1 -7614.794,E2 -7614.794} C_VEL
LIN {X 0,Y 468.848,Z 478.348,A -85,B 0,C 180,E1 -7617.85,E2 -7617.85} C_VEL
LIN {X 0,Y 468.402,Z 486.309,A -85,B 0,C 180,E1 -7620.892,E2 -7620.892} C_VEL
LIN {X 0,Y 468.045,Z 493.882,A -85,B 0,C 180,E1 -7623.707,E2 -7623.707} C_VEL
LIN {X 0,Y 467.735,Z 501.38,A -85,B 0,C 180,E1 -7626.429,E2 -7626.429} C_VEL
LIN {X 0,Y 467.412,Z 509.495,A -85,B 0,C 180,E1 -7629.308,E2 -7629.308} C_VEL
LIN {X 0,Y 467.219,Z 517.321,A -85,B 0,C 180,E1 -7632.039,E2 -7632.039} C_VEL
LIN {X 0,Y 467.098,Z 524.82,A -85,B 0,C 180,E1 -7634.619,E2 -7634.619} C_VEL
LIN {X 0,Y 469.166,Z 540.253,A -85,B 0,C 180,E1 -7635.141,E2 -7635.141} C_VEL
LIN {X 0,Y 469.863,Z 545.783,A -85,B 0,C 180,E1 -7635.38,E2 -7635.38} C_VEL
LIN {X 0,Y 469.379,Z 558.916,A -85,B 0,C 180,E1 -7636.029,E2 -7636.029} C_VEL
LIN {X 0,Y 468.898,Z 570.554,A -85,B 0,C 180,E1 -7636.787,E2 -7636.787} C_VEL
LIN {X 0,Y 468.386,Z 581.578,A -85,B 0,C 180,E1 -7637.699,E2 -7637.699} C_VEL
LIN {X 0,Y 467.928,Z 591.767,A -85,B 0,C 180,E1 -7638.741,E2 -7638.741} C_VEL
LIN {X 0,Y 467.485,Z 600.46,A -85,B 0,C 180,E1 -7639.826,E2 -7639.826} C_VEL
LIN {X 0,Y 467.163,Z 608.914,A -85,B 0,C 180,E1 -7641.13,E2 -7641.13} C_VEL
LIN {X 0,Y 466.928,Z 615.723,A -85,B 0,C 180,E1 -7642.432,E2 -7642.432} C_VEL
LIN {X 0,Y 466.768,Z 621.973,A -85,B 0,C 180,E1 -7643.95,E2 -7643.95} C_VEL
LIN {X 0,Y 466.7,Z 626.022,A -85,B 0,C 180,E1 -7645.249,E2 -7645.249} C_VEL
LIN {X 0,Y 466.73,Z 629.006,A -85,B 0,C 180,E1 -7646.547,E2 -7646.547} C_VEL
LIN {X 0,Y 466.7,Z 630.428,A -85,B 0,C 180,E1 -7647.411,E2 -7647.411} C_VEL
LIN {X 0,Y 466.693,Z 631.429,A -85,B 0,C 180,E1 -7648.274,E2 -7648.274} C_VEL
LIN {X 0,Y 466.62,Z 632.028,A -85,B 0,C 180,E1 -7649.137,E2 -7649.137} C_VEL
LIN {X 0,Y 466.598,Z 632.228,A -85,B 0,C 180,E1 -7650,E2 -7650} C_VEL
